// TIA Portal V16 export
// export: Created 2022-11-17T11:55:09.5879993Z, ExportSetting WithDefaults, DisplayName Totally Integrated Automation Portal, DisplayVersion V16 Update 6, DisplayName TIA Portal Version Control Interface, DisplayVersion V16 Update 2, DisplayName TIA Portal Openness, DisplayVersion V16 Update 6, DisplayName SINAMICS Startdrive Advanced, DisplayVersion V16 Update 5, DisplayName SINAMICS Startdrive G130, G150, S120, S150, SINAMICS MV, S210, DisplayVersion V16 Update 5, DisplayName SINAMICS Startdrive G110M, G120, G120C, G120D, G120P, G115D, DisplayVersion V16 Update 5, DisplayName STEP 7 Professional, DisplayVersion V16 Update 6, DisplayName STEP 7 Safety, DisplayVersion V16, DisplayName WinCC Advanced, DisplayVersion V16 Update 6
FUNCTION "FC23_TopTechnoplat" : Void   // FC23, LAD
TITLE = Top Inside
{ S7_Optimized_Access := 'FALSE' }
VERSION : 0.1
// stored: AutoNumber false, IsIECCheckEnabled false, SetENOAutomatically false, UDAEnableTagReadback false
   VAR_TEMP
      LW4 : Word;
   END_VAR
   VAR_TEMP   // added for the SCL form of the ladder/FBD networks
      _w1 : Bool;
      _w2 : Bool;
   END_VAR
BEGIN

REGION Network 1: Top Out Supp. Out - Signal " Top In Position for Pallet Transfe
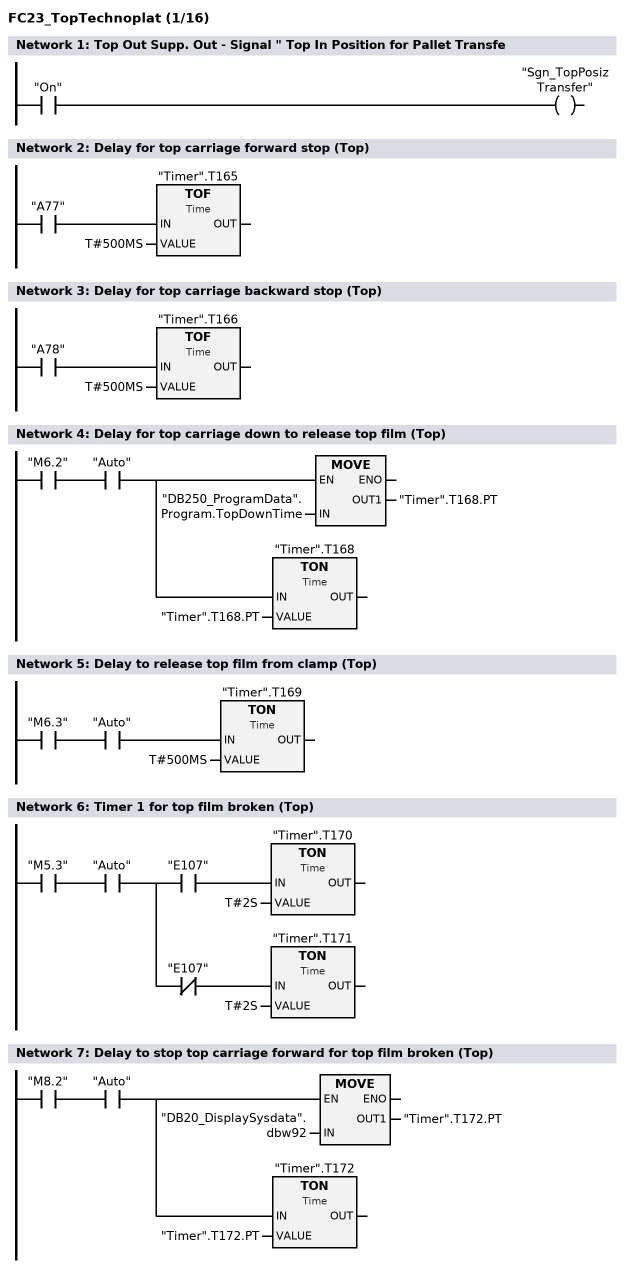
   RUNG wire#powerrail
      Contact( "On" )
      Coil( "Sgn_TopPosizTransfer" )
   END_RUNG
   // the same network as SCL:
   "Sgn_TopPosizTransfer" := "On";
END_REGION

REGION Network 2: Delay for top carriage forward stop (Top)
   "Timer".T165.TOF(IN := "A77", PT := T#500MS);   // TOF coil
END_REGION

REGION Network 3: Delay for top carriage backward stop (Top)
   "Timer".T166.TOF(IN := "A78", PT := T#500MS);   // TOF coil
END_REGION

REGION Network 4: Delay for top carriage down to release top film (Top)
   #_w1 := "M6.2" AND "Auto";
   IF #_w1 THEN "Timer".T168.PT := "DB250_ProgramData".Program.TopDownTime; END_IF;
   "Timer".T168.TON(IN := #_w1, PT := "Timer".T168.PT);   // TON coil
END_REGION

REGION Network 5: Delay to release top film from clamp (Top)
   "Timer".T169.TON(IN := "M6.3" AND "Auto", PT := T#500MS);   // TON coil
END_REGION

REGION Network 6: Timer 1 for top film broken (Top)
   #_w1 := "M5.3" AND "Auto";
   "Timer".T170.TON(IN := #_w1 AND "E107", PT := T#2S);   // TON coil
   "Timer".T171.TON(IN := #_w1 AND NOT "E107", PT := T#2S);   // TON coil
END_REGION

REGION Network 7: Delay to stop top carriage forward for top film broken (Top)
   #_w1 := "M8.2" AND "Auto";
   IF #_w1 THEN "Timer".T172.PT := "DB20_DisplaySysdata".dbw92; END_IF;
   "Timer".T172.TON(IN := #_w1, PT := "Timer".T172.PT);   // TON coil
END_REGION

REGION Network 8: Delay to stop top carriage against vibration (Top)
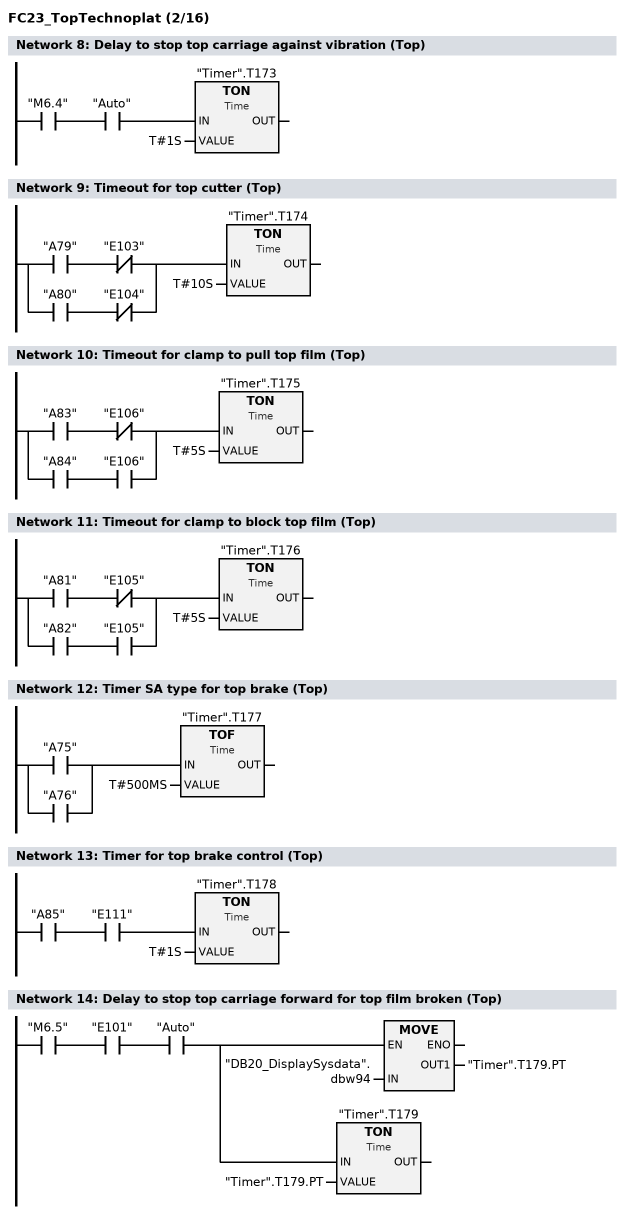
   "Timer".T173.TON(IN := "M6.4" AND "Auto", PT := T#1S);   // TON coil
END_REGION

REGION Network 9: Timeout for top cutter (Top)
   "Timer".T174.TON(IN := ("A79" AND NOT "E103") OR ("A80" AND NOT "E104"), PT := T#10S);   // TON coil
END_REGION

REGION Network 10: Timeout for clamp to pull top film (Top)
   "Timer".T175.TON(IN := ("A83" AND NOT "E106") OR ("A84" AND "E106"), PT := T#5S);   // TON coil
END_REGION

REGION Network 11: Timeout for clamp to block top film (Top)
   "Timer".T176.TON(IN := ("A81" AND NOT "E105") OR ("A82" AND "E105"), PT := T#5S);   // TON coil
END_REGION

REGION Network 12: Timer SA type for top brake (Top)
   "Timer".T177.TOF(IN := "A75" OR "A76", PT := T#500MS);   // TOF coil
END_REGION

REGION Network 13: Timer for top brake control (Top)
   "Timer".T178.TON(IN := "A85" AND "E111", PT := T#1S);   // TON coil
END_REGION

REGION Network 14: Delay to stop top carriage forward for top film broken (Top)
   #_w1 := "M6.5" AND "E101" AND "Auto";
   IF #_w1 THEN "Timer".T179.PT := "DB20_DisplaySysdata".dbw94; END_IF;
   "Timer".T179.TON(IN := #_w1, PT := "Timer".T179.PT);   // TON coil
END_REGION

REGION Network 15: Carriage in position to rotate in medium to wrap top
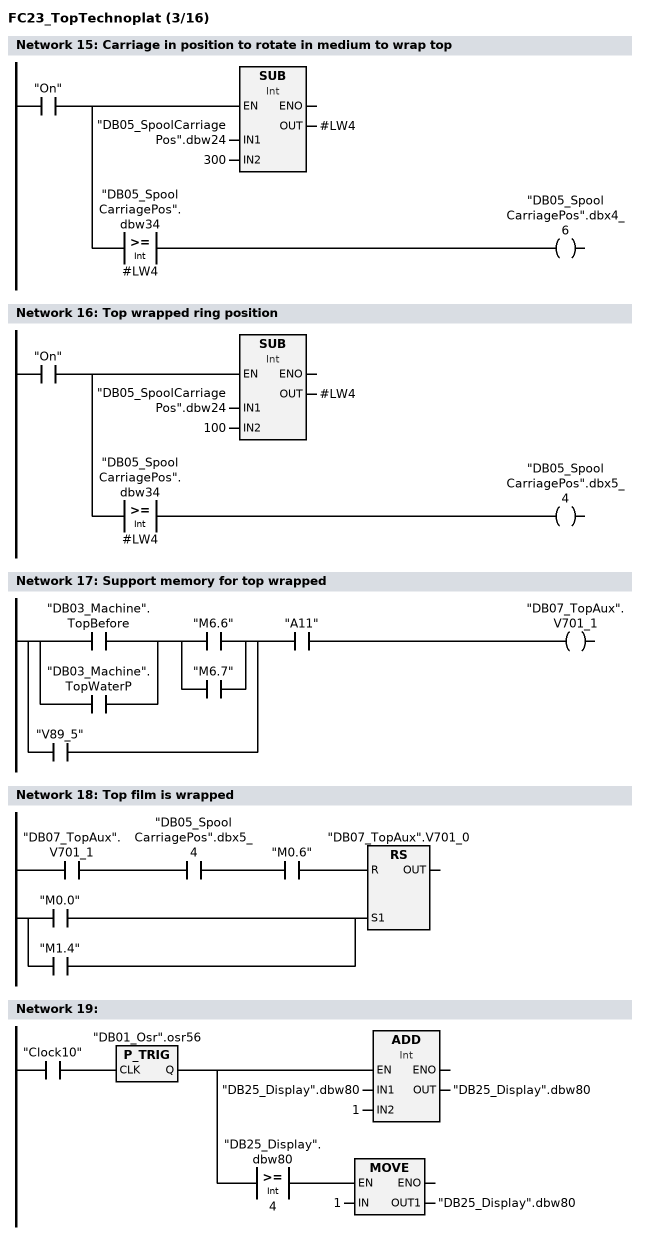
   RUNG wire#powerrail
      Contact( "On" )
      wire#w1
      { S7_Templates := "SrcType := Int"; S7_GenerateENO := "TRUE" } Sub(in1 := "DB05_SpoolCarriagePos".dbw24, in2 := 300, out => #LW4)
   END_RUNG
   RUNG wire#w1
      { S7_Templates := "SrcType := Int" } GE_Contact(in1 := "DB05_SpoolCarriagePos".dbw34, in2 := #LW4)
      Coil( "DB05_SpoolCarriagePos".dbx4_6 )
   END_RUNG
   // the same network as SCL:
   IF "On" THEN #LW4 := "DB05_SpoolCarriagePos".dbw24 - 300; END_IF;
   "DB05_SpoolCarriagePos".dbx4_6 := "On" AND ("DB05_SpoolCarriagePos".dbw34 >= #LW4);
END_REGION

REGION Network 16: Top wrapped ring position
   RUNG wire#powerrail
      Contact( "On" )
      wire#w1
      { S7_Templates := "SrcType := Int"; S7_GenerateENO := "TRUE" } Sub(in1 := "DB05_SpoolCarriagePos".dbw24, in2 := 100, out => #LW4)
   END_RUNG
   RUNG wire#w1
      { S7_Templates := "SrcType := Int" } GE_Contact(in1 := "DB05_SpoolCarriagePos".dbw34, in2 := #LW4)
      Coil( "DB05_SpoolCarriagePos".dbx5_4 )
   END_RUNG
   // the same network as SCL:
   IF "On" THEN #LW4 := "DB05_SpoolCarriagePos".dbw24 - 100; END_IF;
   "DB05_SpoolCarriagePos".dbx5_4 := "On" AND ("DB05_SpoolCarriagePos".dbw34 >= #LW4);
END_REGION

REGION Network 17: Support memory for top wrapped
   RUNG wire#powerrail
      Contact( "DB03_Machine".TopBefore )
      wire#w1
      Contact( "M6.6" )
      wire#w2
      Contact( "A11" )
      Coil( "DB07_TopAux".V701_1 )
   END_RUNG
   RUNG wire#powerrail
      Contact( "DB03_Machine".TopWaterP )
   END_RUNG wire#w1
   RUNG wire#w1
      Contact( "M6.7" )
   END_RUNG wire#w2
   RUNG wire#powerrail
      Contact( "V89_5" )
   END_RUNG wire#w2
   // the same network as SCL:
   "DB07_TopAux".V701_1 := ((("DB03_Machine".TopBefore OR "DB03_Machine".TopWaterP) AND ("M6.6" OR "M6.7")) OR "V89_5") AND "A11";
END_REGION

REGION Network 18: Top film is wrapped
   RUNG wire#powerrail
      Contact( "DB07_TopAux".V701_1 )
      Contact( "DB05_SpoolCarriagePos".dbx5_4 )
      Contact( "M0.6" )
      S_RS(operand := "DB07_TopAux".V701_0, s1 := wire#w1)
   END_RUNG
   RUNG wire#powerrail
      Contact( "M0.0" )
   END_RUNG wire#w1
   RUNG wire#powerrail
      Contact( "M1.4" )
   END_RUNG wire#w1
   // the same network as SCL:
   IF "DB07_TopAux".V701_1 AND "DB05_SpoolCarriagePos".dbx5_4 AND "M0.6" THEN
       "DB07_TopAux".V701_0 := FALSE;   // RS flip-flop
   END_IF;
   IF "M0.0" OR "M1.4" THEN "DB07_TopAux".V701_0 := TRUE; END_IF;
END_REGION

REGION Network 19
   RUNG wire#powerrail
      Contact( "Clock10" )
      P_Trig( "DB01_Osr".osr56 )
      wire#w1
      { S7_Templates := "SrcType := Int"; S7_GenerateENO := "TRUE" } Add(in1 := "DB25_Display".dbw80, in2 := 1, out => "DB25_Display".dbw80)
   END_RUNG
   RUNG wire#w1
      { S7_Templates := "SrcType := Int" } GE_Contact(in1 := "DB25_Display".dbw80, in2 := 4)
      { S7_GenerateENO := "TRUE" } Move(in := 1, out1 => "DB25_Display".dbw80)
   END_RUNG
   // the same network as SCL:
   #_w1 := "Clock10" AND NOT "DB01_Osr".osr56;   // rising edge
   "DB01_Osr".osr56 := "Clock10";
   IF #_w1 THEN "DB25_Display".dbw80 := "DB25_Display".dbw80 + 1; END_IF;
   IF #_w1 AND ("DB25_Display".dbw80 >= 4) THEN "DB25_Display".dbw80 := 1; END_IF;
END_REGION

REGION Network 20: Arm rotation speed: Middle 1 for top
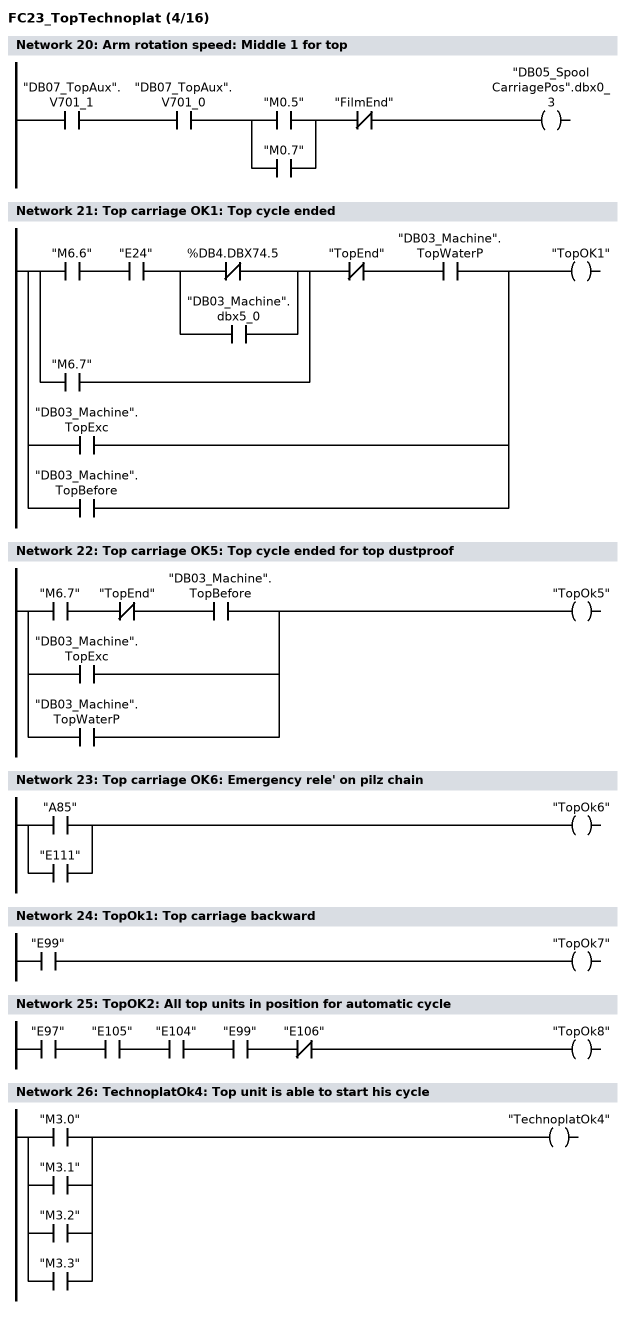
   RUNG wire#powerrail
      Contact( "DB07_TopAux".V701_1 )
      Contact( "DB07_TopAux".V701_0 )
      wire#w1
      Contact( "M0.5" )
      wire#w2
      I_Contact( "FilmEnd" )
      Coil( "DB05_SpoolCarriagePos".dbx0_3 )
   END_RUNG
   RUNG wire#w1
      Contact( "M0.7" )
   END_RUNG wire#w2
   // the same network as SCL:
   "DB05_SpoolCarriagePos".dbx0_3 := "DB07_TopAux".V701_1 AND "DB07_TopAux".V701_0 AND ("M0.5" OR "M0.7") AND NOT "FilmEnd";
END_REGION

REGION Network 21: Top carriage OK1: Top cycle ended
   RUNG wire#powerrail
      Contact( "M6.6" )
      Contact( "E24" )
      wire#w1
      I_Contact( %DB4.DBX74.5 )
      wire#w2
      I_Contact( "TopEnd" )
      Contact( "DB03_Machine".TopWaterP )
      wire#w3
      Coil( "TopOK1" )
   END_RUNG
   RUNG wire#w1
      Contact( "DB03_Machine".dbx5_0 )
   END_RUNG wire#w2
   RUNG wire#powerrail
      Contact( "M6.7" )
   END_RUNG wire#w2
   RUNG wire#powerrail
      Contact( "DB03_Machine".TopExc )
   END_RUNG wire#w3
   RUNG wire#powerrail
      Contact( "DB03_Machine".TopBefore )
   END_RUNG wire#w3
   // the same network as SCL:
   "TopOK1" := ((("M6.6" AND "E24" AND (NOT %DB4.DBX74.5 OR "DB03_Machine".dbx5_0)) OR "M6.7") AND NOT "TopEnd" AND "DB03_Machine".TopWaterP) OR "DB03_Machine".TopExc OR "DB03_Machine".TopBefore;
END_REGION

REGION Network 22: Top carriage OK5: Top cycle ended for top dustproof
   RUNG wire#powerrail
      Contact( "M6.7" )
      I_Contact( "TopEnd" )
      Contact( "DB03_Machine".TopBefore )
      wire#w1
      Coil( "TopOk5" )
   END_RUNG
   RUNG wire#powerrail
      Contact( "DB03_Machine".TopExc )
   END_RUNG wire#w1
   RUNG wire#powerrail
      Contact( "DB03_Machine".TopWaterP )
   END_RUNG wire#w1
   // the same network as SCL:
   "TopOk5" := ("M6.7" AND NOT "TopEnd" AND "DB03_Machine".TopBefore) OR "DB03_Machine".TopExc OR "DB03_Machine".TopWaterP;
END_REGION

REGION Network 23: Top carriage OK6: Emergency rele' on pilz chain
   RUNG wire#powerrail
      Contact( "A85" )
      wire#w1
      Coil( "TopOk6" )
   END_RUNG
   RUNG wire#powerrail
      Contact( "E111" )
   END_RUNG wire#w1
   // the same network as SCL:
   "TopOk6" := "A85" OR "E111";
END_REGION

REGION Network 24: TopOk1: Top carriage backward
   RUNG wire#powerrail
      Contact( "E99" )
      Coil( "TopOk7" )
   END_RUNG
   // the same network as SCL:
   "TopOk7" := "E99";
END_REGION

REGION Network 25: TopOK2: All top units in position for automatic cycle
   RUNG wire#powerrail
      Contact( "E97" )
      Contact( "E105" )
      Contact( "E104" )
      Contact( "E99" )
      I_Contact( "E106" )
      Coil( "TopOk8" )
   END_RUNG
   // the same network as SCL:
   "TopOk8" := "E97" AND "E105" AND "E104" AND "E99" AND NOT "E106";
END_REGION

REGION Network 26: TechnoplatOk4: Top unit is able to start his cycle
   RUNG wire#powerrail
      Contact( "M3.0" )
      wire#w1
      Coil( "TechnoplatOk4" )
   END_RUNG
   RUNG wire#powerrail
      Contact( "M3.1" )
   END_RUNG wire#w1
   RUNG wire#powerrail
      Contact( "M3.2" )
   END_RUNG wire#w1
   RUNG wire#powerrail
      Contact( "M3.3" )
   END_RUNG wire#w1
   // the same network as SCL:
   "TechnoplatOk4" := "M3.0" OR "M3.1" OR "M3.2" OR "M3.3";
END_REGION

REGION Network 27: Top film ended or broken
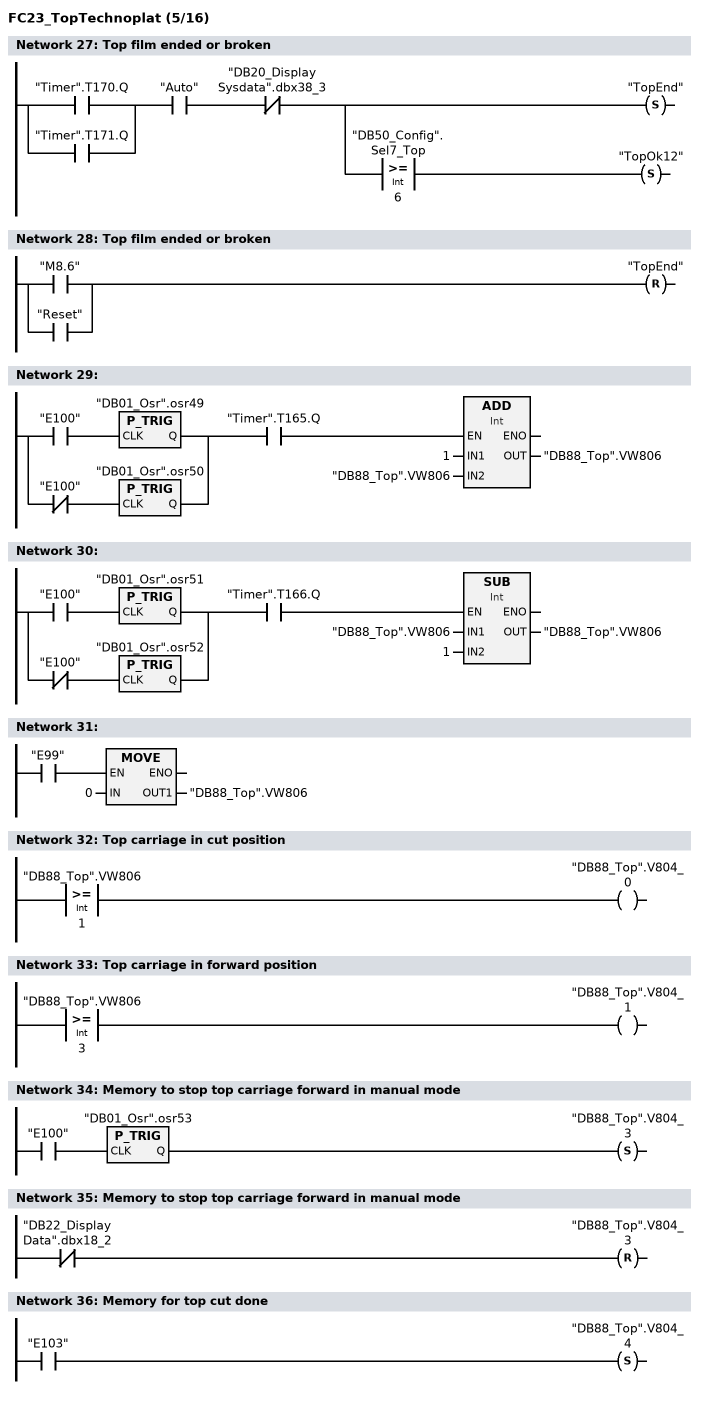
   RUNG wire#powerrail
      Contact( "Timer".T170.Q )
      wire#w1
      Contact( "Auto" )
      I_Contact( "DB20_DisplaySysdata".dbx38_3 )
      wire#w2
      S_Coil( "TopEnd" )
   END_RUNG
   RUNG wire#powerrail
      Contact( "Timer".T171.Q )
   END_RUNG wire#w1
   RUNG wire#w2
      { S7_Templates := "SrcType := Int" } GE_Contact(in1 := "DB50_Config".Sel7_Top, in2 := 6)
      S_Coil( "TopOk12" )
   END_RUNG
   // the same network as SCL:
   #_w1 := ("Timer".T170.Q OR "Timer".T171.Q) AND "Auto" AND NOT "DB20_DisplaySysdata".dbx38_3;
   IF #_w1 THEN "TopEnd" := TRUE; END_IF;
   IF #_w1 AND ("DB50_Config".Sel7_Top >= 6) THEN "TopOk12" := TRUE; END_IF;
END_REGION

REGION Network 28: Top film ended or broken
   RUNG wire#powerrail
      Contact( "M8.6" )
      wire#w1
      R_Coil( "TopEnd" )
   END_RUNG
   RUNG wire#powerrail
      Contact( "Reset" )
   END_RUNG wire#w1
   // the same network as SCL:
   IF "M8.6" OR "Reset" THEN "TopEnd" := FALSE; END_IF;
END_REGION

REGION Network 29
   RUNG wire#powerrail
      Contact( "E100" )
      P_Trig( "DB01_Osr".osr49 )
      wire#w1
      Contact( "Timer".T165.Q )
      { S7_Templates := "SrcType := Int"; S7_GenerateENO := "TRUE" } Add(in1 := 1, in2 := "DB88_Top".VW806, out => "DB88_Top".VW806)
   END_RUNG
   RUNG wire#powerrail
      I_Contact( "E100" )
      P_Trig( "DB01_Osr".osr50 )
   END_RUNG wire#w1
   // the same network as SCL:
   #_w1 := "E100" AND NOT "DB01_Osr".osr49;   // rising edge
   "DB01_Osr".osr49 := "E100";
   #_w2 := NOT "E100" AND NOT "DB01_Osr".osr50;   // rising edge
   "DB01_Osr".osr50 := NOT "E100";
   IF (#_w1 OR #_w2) AND "Timer".T165.Q THEN "DB88_Top".VW806 := 1 + "DB88_Top".VW806; END_IF;
END_REGION

REGION Network 30
   RUNG wire#powerrail
      Contact( "E100" )
      P_Trig( "DB01_Osr".osr51 )
      wire#w1
      Contact( "Timer".T166.Q )
      { S7_Templates := "SrcType := Int"; S7_GenerateENO := "TRUE" } Sub(in1 := "DB88_Top".VW806, in2 := 1, out => "DB88_Top".VW806)
   END_RUNG
   RUNG wire#powerrail
      I_Contact( "E100" )
      P_Trig( "DB01_Osr".osr52 )
   END_RUNG wire#w1
   // the same network as SCL:
   #_w1 := "E100" AND NOT "DB01_Osr".osr51;   // rising edge
   "DB01_Osr".osr51 := "E100";
   #_w2 := NOT "E100" AND NOT "DB01_Osr".osr52;   // rising edge
   "DB01_Osr".osr52 := NOT "E100";
   IF (#_w1 OR #_w2) AND "Timer".T166.Q THEN "DB88_Top".VW806 := "DB88_Top".VW806 - 1; END_IF;
END_REGION

REGION Network 31
   RUNG wire#powerrail
      Contact( "E99" )
      { S7_GenerateENO := "TRUE" } Move(in := 0, out1 => "DB88_Top".VW806)
   END_RUNG
   // the same network as SCL:
   IF "E99" THEN "DB88_Top".VW806 := 0; END_IF;
END_REGION

REGION Network 32: Top carriage in cut position
   RUNG wire#powerrail
      { S7_Templates := "SrcType := Int" } GE_Contact(in1 := "DB88_Top".VW806, in2 := 1)
      Coil( "DB88_Top".V804_0 )
   END_RUNG
   // the same network as SCL:
   "DB88_Top".V804_0 := "DB88_Top".VW806 >= 1;
END_REGION

REGION Network 33: Top carriage in forward position
   RUNG wire#powerrail
      { S7_Templates := "SrcType := Int" } GE_Contact(in1 := "DB88_Top".VW806, in2 := 3)
      Coil( "DB88_Top".V804_1 )
   END_RUNG
   // the same network as SCL:
   "DB88_Top".V804_1 := "DB88_Top".VW806 >= 3;
END_REGION

REGION Network 34: Memory to stop top carriage forward in manual mode
   RUNG wire#powerrail
      Contact( "E100" )
      P_Trig( "DB01_Osr".osr53 )
      S_Coil( "DB88_Top".V804_3 )
   END_RUNG
   // the same network as SCL:
   #_w1 := "E100" AND NOT "DB01_Osr".osr53;   // rising edge
   "DB01_Osr".osr53 := "E100";
   IF #_w1 THEN "DB88_Top".V804_3 := TRUE; END_IF;
END_REGION

REGION Network 35: Memory to stop top carriage forward in manual mode
   RUNG wire#powerrail
      I_Contact( "DB22_DisplayData".dbx18_2 )
      R_Coil( "DB88_Top".V804_3 )
   END_RUNG
   // the same network as SCL:
   IF NOT "DB22_DisplayData".dbx18_2 THEN "DB88_Top".V804_3 := FALSE; END_IF;
END_REGION

REGION Network 36: Memory for top cut done
   RUNG wire#powerrail
      Contact( "E103" )
      S_Coil( "DB88_Top".V804_4 )
   END_RUNG
   // the same network as SCL:
   IF "E103" THEN "DB88_Top".V804_4 := TRUE; END_IF;
END_REGION

REGION Network 37: Memory for top cut done
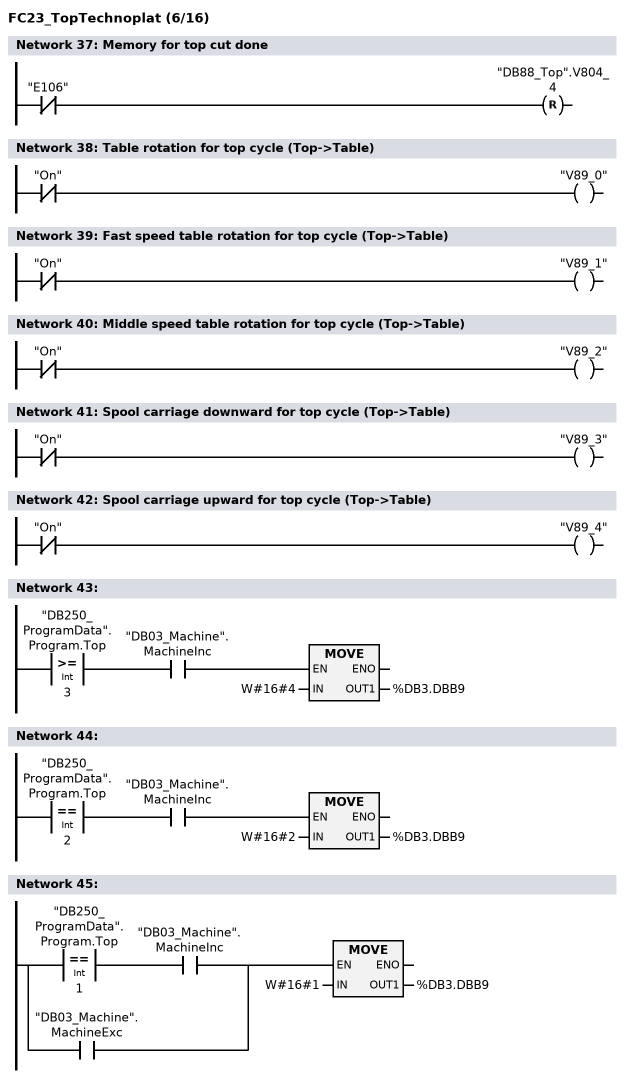
   RUNG wire#powerrail
      I_Contact( "E106" )
      R_Coil( "DB88_Top".V804_4 )
   END_RUNG
   // the same network as SCL:
   IF NOT "E106" THEN "DB88_Top".V804_4 := FALSE; END_IF;
END_REGION

REGION Network 38: Table rotation for top cycle (Top->Table)
   RUNG wire#powerrail
      I_Contact( "On" )
      Coil( "V89_0" )
   END_RUNG
   // the same network as SCL:
   "V89_0" := NOT "On";
END_REGION

REGION Network 39: Fast speed table rotation for top cycle (Top->Table)
   RUNG wire#powerrail
      I_Contact( "On" )
      Coil( "V89_1" )
   END_RUNG
   // the same network as SCL:
   "V89_1" := NOT "On";
END_REGION

REGION Network 40: Middle speed table rotation for top cycle (Top->Table)
   RUNG wire#powerrail
      I_Contact( "On" )
      Coil( "V89_2" )
   END_RUNG
   // the same network as SCL:
   "V89_2" := NOT "On";
END_REGION

REGION Network 41: Spool carriage downward for top cycle (Top->Table)
   RUNG wire#powerrail
      I_Contact( "On" )
      Coil( "V89_3" )
   END_RUNG
   // the same network as SCL:
   "V89_3" := NOT "On";
END_REGION

REGION Network 42: Spool carriage upward for top cycle (Top->Table)
   RUNG wire#powerrail
      I_Contact( "On" )
      Coil( "V89_4" )
   END_RUNG
   // the same network as SCL:
   "V89_4" := NOT "On";
END_REGION

REGION Network 43
   RUNG wire#powerrail
      { S7_Templates := "SrcType := Int" } GE_Contact(in1 := "DB250_ProgramData".Program.Top, in2 := 3)
      Contact( "DB03_Machine".MachineInc )
      { S7_GenerateENO := "TRUE" } Move(in := W#16#4, out1 => %DB3.DBB9)
   END_RUNG
   // the same network as SCL:
   IF ("DB250_ProgramData".Program.Top >= 3) AND "DB03_Machine".MachineInc THEN %DB3.DBB9 := W#16#4; END_IF;
END_REGION

REGION Network 44
   RUNG wire#powerrail
      { S7_Templates := "SrcType := Int" } EQ_Contact(in1 := "DB250_ProgramData".Program.Top, in2 := 2)
      Contact( "DB03_Machine".MachineInc )
      { S7_GenerateENO := "TRUE" } Move(in := W#16#2, out1 => %DB3.DBB9)
   END_RUNG
   // the same network as SCL:
   IF ("DB250_ProgramData".Program.Top = 2) AND "DB03_Machine".MachineInc THEN %DB3.DBB9 := W#16#2; END_IF;
END_REGION

REGION Network 45
   RUNG wire#powerrail
      { S7_Templates := "SrcType := Int" } EQ_Contact(in1 := "DB250_ProgramData".Program.Top, in2 := 1)
      Contact( "DB03_Machine".MachineInc )
      wire#w1
      { S7_GenerateENO := "TRUE" } Move(in := W#16#1, out1 => %DB3.DBB9)
   END_RUNG
   RUNG wire#powerrail
      Contact( "DB03_Machine".MachineExc )
   END_RUNG wire#w1
   // the same network as SCL:
   IF (("DB250_ProgramData".Program.Top = 1) AND "DB03_Machine".MachineInc) OR "DB03_Machine".MachineExc THEN
       %DB3.DBB9 := W#16#1;
   END_IF;
END_REGION

REGION Network 46: Wrapping cycle: After this step top waterproof
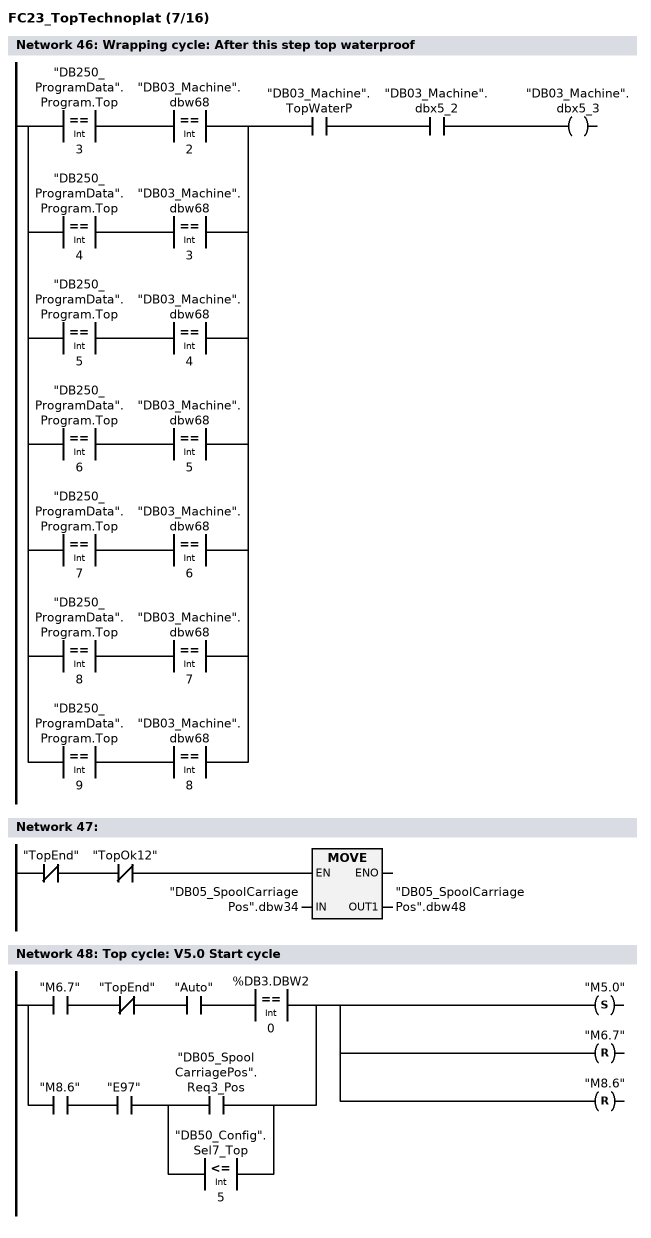
   RUNG wire#powerrail
      { S7_Templates := "SrcType := Int" } EQ_Contact(in1 := "DB250_ProgramData".Program.Top, in2 := 3)
      { S7_Templates := "SrcType := Int" } EQ_Contact(in1 := "DB03_Machine".dbw68, in2 := 2)
      wire#w1
      Contact( "DB03_Machine".TopWaterP )
      Contact( "DB03_Machine".dbx5_2 )
      Coil( "DB03_Machine".dbx5_3 )
   END_RUNG
   RUNG wire#powerrail
      { S7_Templates := "SrcType := Int" } EQ_Contact(in1 := "DB250_ProgramData".Program.Top, in2 := 4)
      { S7_Templates := "SrcType := Int" } EQ_Contact(in1 := "DB03_Machine".dbw68, in2 := 3)
   END_RUNG wire#w1
   RUNG wire#powerrail
      { S7_Templates := "SrcType := Int" } EQ_Contact(in1 := "DB250_ProgramData".Program.Top, in2 := 5)
      { S7_Templates := "SrcType := Int" } EQ_Contact(in1 := "DB03_Machine".dbw68, in2 := 4)
   END_RUNG wire#w1
   RUNG wire#powerrail
      { S7_Templates := "SrcType := Int" } EQ_Contact(in1 := "DB250_ProgramData".Program.Top, in2 := 6)
      { S7_Templates := "SrcType := Int" } EQ_Contact(in1 := "DB03_Machine".dbw68, in2 := 5)
   END_RUNG wire#w1
   RUNG wire#powerrail
      { S7_Templates := "SrcType := Int" } EQ_Contact(in1 := "DB250_ProgramData".Program.Top, in2 := 7)
      { S7_Templates := "SrcType := Int" } EQ_Contact(in1 := "DB03_Machine".dbw68, in2 := 6)
   END_RUNG wire#w1
   RUNG wire#powerrail
      { S7_Templates := "SrcType := Int" } EQ_Contact(in1 := "DB250_ProgramData".Program.Top, in2 := 8)
      { S7_Templates := "SrcType := Int" } EQ_Contact(in1 := "DB03_Machine".dbw68, in2 := 7)
   END_RUNG wire#w1
   RUNG wire#powerrail
      { S7_Templates := "SrcType := Int" } EQ_Contact(in1 := "DB250_ProgramData".Program.Top, in2 := 9)
      { S7_Templates := "SrcType := Int" } EQ_Contact(in1 := "DB03_Machine".dbw68, in2 := 8)
   END_RUNG wire#w1
   // the same network as SCL:
   "DB03_Machine".dbx5_3 := ((("DB250_ProgramData".Program.Top = 3) AND ("DB03_Machine".dbw68 = 2)) OR (("DB250_ProgramData".Program.Top = 4) AND ("DB03_Machine".dbw68 = 3)) OR (("DB250_ProgramData".Program.Top = 5) AND ("DB03_Machine".dbw68 = 4)) OR (("DB250_ProgramData".Program.Top = 6) AND ("DB03_Machine".dbw68 = 5)) OR (("DB250_ProgramData".Program.Top = 7) AND ("DB03_Machine".dbw68 = 6)) OR (("DB250_ProgramData".Program.Top = 8) AND ("DB03_Machine".dbw68 = 7)) OR (("DB250_ProgramData".Program.Top = 9) AND ("DB03_Machine".dbw68 = 8))) AND "DB03_Machine".TopWaterP AND "DB03_Machine".dbx5_2;
END_REGION

REGION Network 47
   RUNG wire#powerrail
      I_Contact( "TopEnd" )
      I_Contact( "TopOk12" )
      { S7_GenerateENO := "TRUE" } Move(in := "DB05_SpoolCarriagePos".dbw34, out1 => "DB05_SpoolCarriagePos".dbw48)
   END_RUNG
   // the same network as SCL:
   IF NOT "TopEnd" AND NOT "TopOk12" THEN
       "DB05_SpoolCarriagePos".dbw48 := "DB05_SpoolCarriagePos".dbw34;
   END_IF;
END_REGION

REGION Network 48: Top cycle: V5.0 Start cycle
   RUNG wire#powerrail
      Contact( "M6.7" )
      I_Contact( "TopEnd" )
      Contact( "Auto" )
      { S7_Templates := "SrcType := Int" } EQ_Contact(in1 := %DB3.DBW2, in2 := 0)
      wire#w1
      S_Coil( "M5.0" )
   END_RUNG
   RUNG wire#powerrail
      Contact( "M8.6" )
      Contact( "E97" )
      wire#w2
      Contact( "DB05_SpoolCarriagePos".Req3_Pos )
   END_RUNG wire#w1
   RUNG wire#w2
      { S7_Templates := "SrcType := Int" } LE_Contact(in1 := "DB50_Config".Sel7_Top, in2 := 5)
   END_RUNG wire#w1
   RUNG wire#w1
      R_Coil( "M6.7" )
   END_RUNG
   RUNG wire#w1
      R_Coil( "M8.6" )
   END_RUNG
   // the same network as SCL:
   IF ("M6.7" AND NOT "TopEnd" AND "Auto" AND (%DB3.DBW2 = 0)) OR ("M8.6" AND "E97" AND ("DB05_SpoolCarriagePos".Req3_Pos OR ("DB50_Config".Sel7_Top <= 5))) THEN
       "M5.0" := TRUE;
   END_IF;
   #_w1 := ("M6.7" AND NOT "TopEnd" AND "Auto" AND (%DB3.DBW2 = 0)) OR ("M8.6" AND "E97" AND ("DB05_SpoolCarriagePos".Req3_Pos OR ("DB50_Config".Sel7_Top <= 5)));
   IF #_w1 THEN
       "M6.7" := FALSE;
       "M8.6" := FALSE;
   END_IF;
END_REGION

REGION Network 49: Top cycle: V5.1 Closing clamp to pull top film
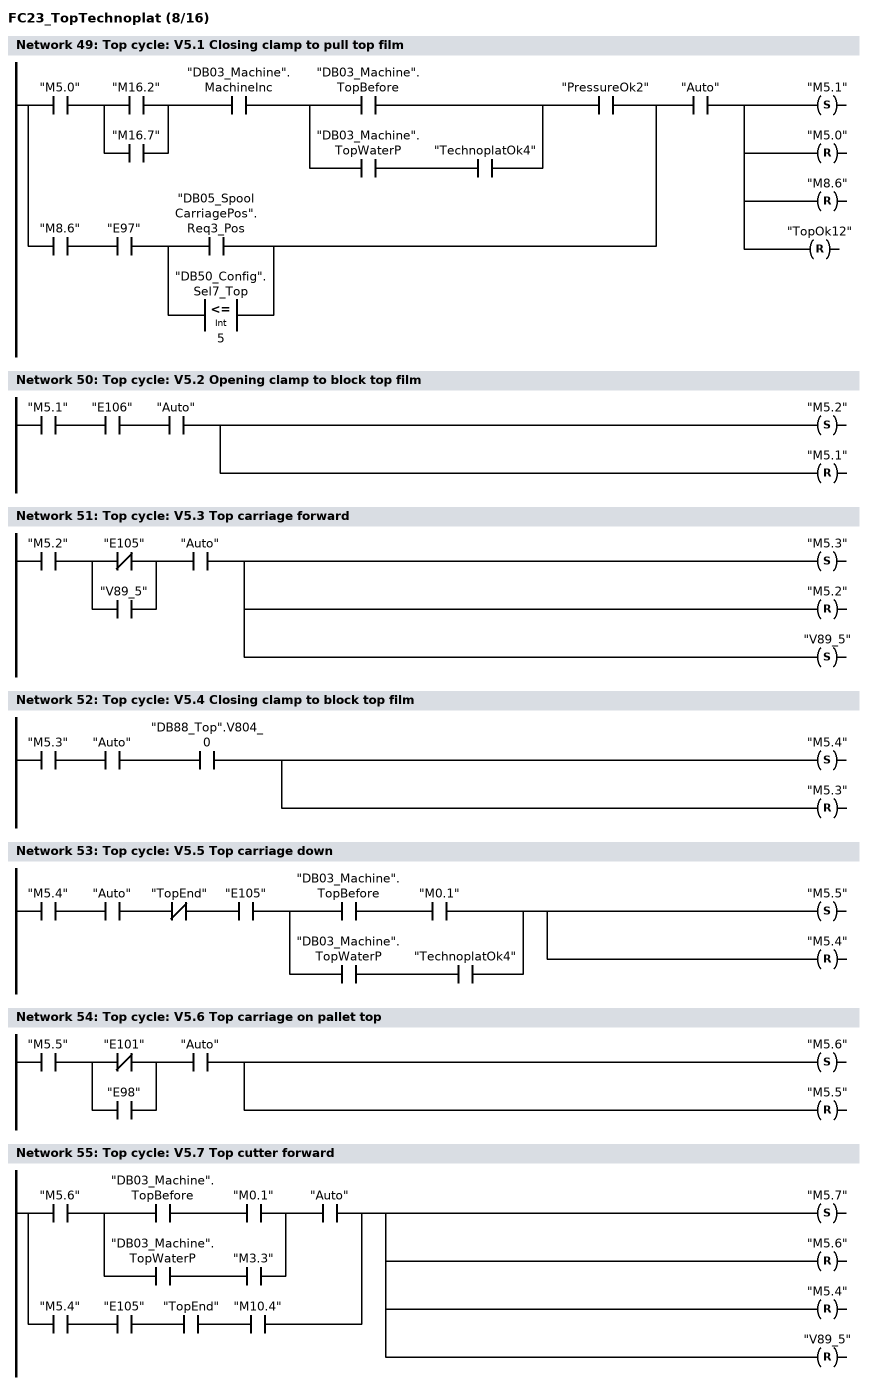
   RUNG wire#powerrail
      Contact( "M5.0" )
      wire#w1
      Contact( "M16.2" )
      wire#w2
      Contact( "DB03_Machine".MachineInc )
      wire#w3
      Contact( "DB03_Machine".TopBefore )
      wire#w4
      Contact( "PressureOk2" )
      wire#w5
      Contact( "Auto" )
      wire#w7
      S_Coil( "M5.1" )
   END_RUNG
   RUNG wire#w1
      Contact( "M16.7" )
   END_RUNG wire#w2
   RUNG wire#w3
      Contact( "DB03_Machine".TopWaterP )
      Contact( "TechnoplatOk4" )
   END_RUNG wire#w4
   RUNG wire#powerrail
      Contact( "M8.6" )
      Contact( "E97" )
      wire#w6
      Contact( "DB05_SpoolCarriagePos".Req3_Pos )
   END_RUNG wire#w5
   RUNG wire#w6
      { S7_Templates := "SrcType := Int" } LE_Contact(in1 := "DB50_Config".Sel7_Top, in2 := 5)
   END_RUNG wire#w5
   RUNG wire#w7
      R_Coil( "M5.0" )
   END_RUNG
   RUNG wire#w7
      R_Coil( "M8.6" )
   END_RUNG
   RUNG wire#w7
      R_Coil( "TopOk12" )
   END_RUNG
   // the same network as SCL:
   IF (("M5.0" AND ("M16.2" OR "M16.7") AND "DB03_Machine".MachineInc AND ("DB03_Machine".TopBefore OR ("DB03_Machine".TopWaterP AND "TechnoplatOk4")) AND "PressureOk2") OR ("M8.6" AND "E97" AND ("DB05_SpoolCarriagePos".Req3_Pos OR ("DB50_Config".Sel7_Top <= 5)))) AND "Auto" THEN
       "M5.1" := TRUE;
   END_IF;
   #_w1 := (("M5.0" AND ("M16.2" OR "M16.7") AND "DB03_Machine".MachineInc AND ("DB03_Machine".TopBefore OR ("DB03_Machine".TopWaterP AND "TechnoplatOk4")) AND "PressureOk2") OR ("M8.6" AND "E97" AND ("DB05_SpoolCarriagePos".Req3_Pos OR ("DB50_Config".Sel7_Top <= 5)))) AND "Auto";
   IF #_w1 THEN
       "M5.0" := FALSE;
       "M8.6" := FALSE;
       "TopOk12" := FALSE;
   END_IF;
END_REGION

REGION Network 50: Top cycle: V5.2 Opening clamp to block top film
   RUNG wire#powerrail
      Contact( "M5.1" )
      Contact( "E106" )
      Contact( "Auto" )
      wire#w1
      S_Coil( "M5.2" )
   END_RUNG
   RUNG wire#w1
      R_Coil( "M5.1" )
   END_RUNG
   // the same network as SCL:
   IF "M5.1" AND "E106" AND "Auto" THEN
       "M5.2" := TRUE;
       "M5.1" := FALSE;
   END_IF;
END_REGION

REGION Network 51: Top cycle: V5.3 Top carriage forward
   RUNG wire#powerrail
      Contact( "M5.2" )
      wire#w1
      I_Contact( "E105" )
      wire#w2
      Contact( "Auto" )
      wire#w3
      S_Coil( "M5.3" )
   END_RUNG
   RUNG wire#w1
      Contact( "V89_5" )
   END_RUNG wire#w2
   RUNG wire#w3
      R_Coil( "M5.2" )
   END_RUNG
   RUNG wire#w3
      S_Coil( "V89_5" )
   END_RUNG
   // the same network as SCL:
   IF "M5.2" AND (NOT "E105" OR "V89_5") AND "Auto" THEN "M5.3" := TRUE; END_IF;
   #_w1 := "M5.2" AND (NOT "E105" OR "V89_5") AND "Auto";
   IF #_w1 THEN
       "M5.2" := FALSE;
       "V89_5" := TRUE;
   END_IF;
END_REGION

REGION Network 52: Top cycle: V5.4 Closing clamp to block top film
   RUNG wire#powerrail
      Contact( "M5.3" )
      Contact( "Auto" )
      Contact( "DB88_Top".V804_0 )
      wire#w1
      S_Coil( "M5.4" )
   END_RUNG
   RUNG wire#w1
      R_Coil( "M5.3" )
   END_RUNG
   // the same network as SCL:
   IF "M5.3" AND "Auto" AND "DB88_Top".V804_0 THEN
       "M5.4" := TRUE;
       "M5.3" := FALSE;
   END_IF;
END_REGION

REGION Network 53: Top cycle: V5.5 Top carriage down
   RUNG wire#powerrail
      Contact( "M5.4" )
      Contact( "Auto" )
      I_Contact( "TopEnd" )
      Contact( "E105" )
      wire#w1
      Contact( "DB03_Machine".TopBefore )
      Contact( "M0.1" )
      wire#w2
      S_Coil( "M5.5" )
   END_RUNG
   RUNG wire#w1
      Contact( "DB03_Machine".TopWaterP )
      Contact( "TechnoplatOk4" )
   END_RUNG wire#w2
   RUNG wire#w2
      R_Coil( "M5.4" )
   END_RUNG
   // the same network as SCL:
   IF "M5.4" AND "Auto" AND NOT "TopEnd" AND "E105" AND (("DB03_Machine".TopBefore AND "M0.1") OR ("DB03_Machine".TopWaterP AND "TechnoplatOk4")) THEN
       "M5.5" := TRUE;
       "M5.4" := FALSE;
   END_IF;
END_REGION

REGION Network 54: Top cycle: V5.6 Top carriage on pallet top
   RUNG wire#powerrail
      Contact( "M5.5" )
      wire#w1
      I_Contact( "E101" )
      wire#w2
      Contact( "Auto" )
      wire#w3
      S_Coil( "M5.6" )
   END_RUNG
   RUNG wire#w1
      Contact( "E98" )
   END_RUNG wire#w2
   RUNG wire#w3
      R_Coil( "M5.5" )
   END_RUNG
   // the same network as SCL:
   IF "M5.5" AND (NOT "E101" OR "E98") AND "Auto" THEN
       "M5.6" := TRUE;
       "M5.5" := FALSE;
   END_IF;
END_REGION

REGION Network 55: Top cycle: V5.7 Top cutter forward
   RUNG wire#powerrail
      Contact( "M5.6" )
      wire#w1
      Contact( "DB03_Machine".TopBefore )
      Contact( "M0.1" )
      wire#w2
      Contact( "Auto" )
      wire#w3
      S_Coil( "M5.7" )
   END_RUNG
   RUNG wire#w1
      Contact( "DB03_Machine".TopWaterP )
      Contact( "M3.3" )
   END_RUNG wire#w2
   RUNG wire#powerrail
      Contact( "M5.4" )
      Contact( "E105" )
      Contact( "TopEnd" )
      Contact( "M10.4" )
   END_RUNG wire#w3
   RUNG wire#w3
      R_Coil( "M5.6" )
   END_RUNG
   RUNG wire#w3
      R_Coil( "M5.4" )
   END_RUNG
   RUNG wire#w3
      R_Coil( "V89_5" )
   END_RUNG
   // the same network as SCL:
   IF ("M5.6" AND (("DB03_Machine".TopBefore AND "M0.1") OR ("DB03_Machine".TopWaterP AND "M3.3")) AND "Auto") OR ("M5.4" AND "E105" AND "TopEnd" AND "M10.4") THEN
       "M5.7" := TRUE;
   END_IF;
   #_w1 := ("M5.6" AND (("DB03_Machine".TopBefore AND "M0.1") OR ("DB03_Machine".TopWaterP AND "M3.3")) AND "Auto") OR ("M5.4" AND "E105" AND "TopEnd" AND "M10.4");
   IF #_w1 THEN
       "M5.6" := FALSE;
       "M5.4" := FALSE;
       "V89_5" := FALSE;
   END_IF;
END_REGION

REGION Network 56: Top cycle: M6.0 Start cycle
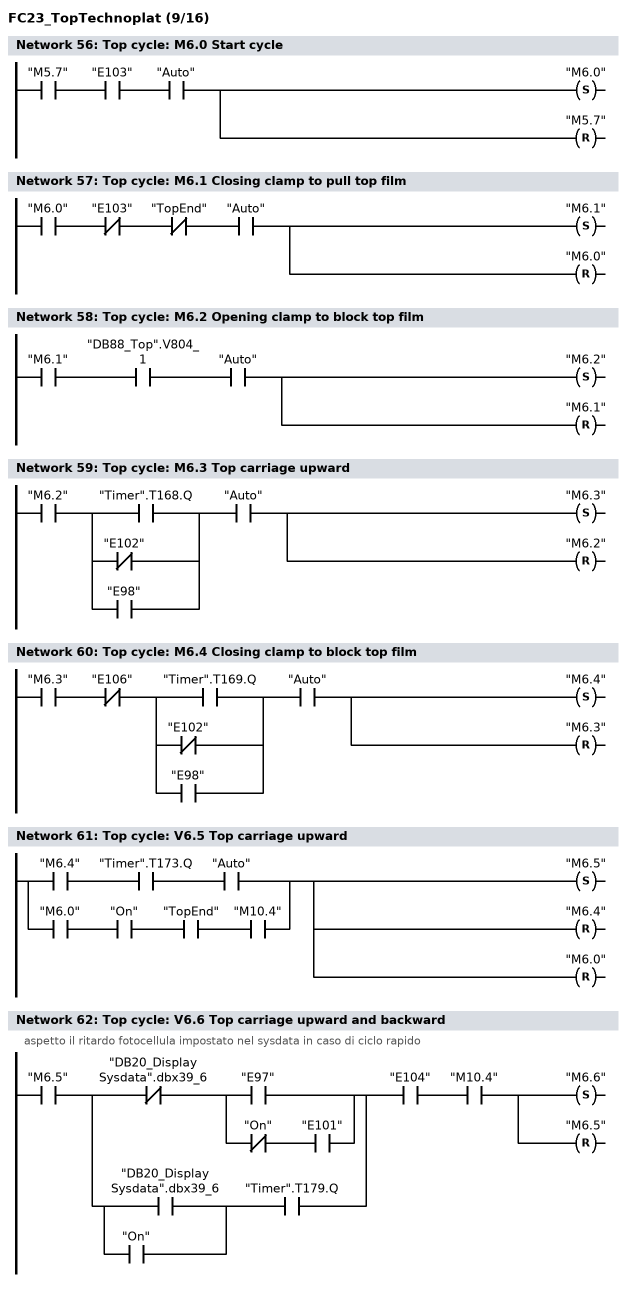
   RUNG wire#powerrail
      Contact( "M5.7" )
      Contact( "E103" )
      Contact( "Auto" )
      wire#w1
      S_Coil( "M6.0" )
   END_RUNG
   RUNG wire#w1
      R_Coil( "M5.7" )
   END_RUNG
   // the same network as SCL:
   IF "M5.7" AND "E103" AND "Auto" THEN
       "M6.0" := TRUE;
       "M5.7" := FALSE;
   END_IF;
END_REGION

REGION Network 57: Top cycle: M6.1 Closing clamp to pull top film
   RUNG wire#powerrail
      Contact( "M6.0" )
      I_Contact( "E103" )
      I_Contact( "TopEnd" )
      Contact( "Auto" )
      wire#w1
      S_Coil( "M6.1" )
   END_RUNG
   RUNG wire#w1
      R_Coil( "M6.0" )
   END_RUNG
   // the same network as SCL:
   IF "M6.0" AND NOT "E103" AND NOT "TopEnd" AND "Auto" THEN
       "M6.1" := TRUE;
       "M6.0" := FALSE;
   END_IF;
END_REGION

REGION Network 58: Top cycle: M6.2 Opening clamp to block top film
   RUNG wire#powerrail
      Contact( "M6.1" )
      Contact( "DB88_Top".V804_1 )
      Contact( "Auto" )
      wire#w1
      S_Coil( "M6.2" )
   END_RUNG
   RUNG wire#w1
      R_Coil( "M6.1" )
   END_RUNG
   // the same network as SCL:
   IF "M6.1" AND "DB88_Top".V804_1 AND "Auto" THEN
       "M6.2" := TRUE;
       "M6.1" := FALSE;
   END_IF;
END_REGION

REGION Network 59: Top cycle: M6.3 Top carriage upward
   RUNG wire#powerrail
      Contact( "M6.2" )
      wire#w1
      Contact( "Timer".T168.Q )
      wire#w2
      Contact( "Auto" )
      wire#w3
      S_Coil( "M6.3" )
   END_RUNG
   RUNG wire#w1
      I_Contact( "E102" )
   END_RUNG wire#w2
   RUNG wire#w1
      Contact( "E98" )
   END_RUNG wire#w2
   RUNG wire#w3
      R_Coil( "M6.2" )
   END_RUNG
   // the same network as SCL:
   IF "M6.2" AND ("Timer".T168.Q OR NOT "E102" OR "E98") AND "Auto" THEN
       "M6.3" := TRUE;
       "M6.2" := FALSE;
   END_IF;
END_REGION

REGION Network 60: Top cycle: M6.4 Closing clamp to block top film
   RUNG wire#powerrail
      Contact( "M6.3" )
      I_Contact( "E106" )
      wire#w1
      Contact( "Timer".T169.Q )
      wire#w2
      Contact( "Auto" )
      wire#w3
      S_Coil( "M6.4" )
   END_RUNG
   RUNG wire#w1
      I_Contact( "E102" )
   END_RUNG wire#w2
   RUNG wire#w1
      Contact( "E98" )
   END_RUNG wire#w2
   RUNG wire#w3
      R_Coil( "M6.3" )
   END_RUNG
   // the same network as SCL:
   IF "M6.3" AND NOT "E106" AND ("Timer".T169.Q OR NOT "E102" OR "E98") AND "Auto" THEN
       "M6.4" := TRUE;
       "M6.3" := FALSE;
   END_IF;
END_REGION

REGION Network 61: Top cycle: V6.5 Top carriage upward
   RUNG wire#powerrail
      Contact( "M6.4" )
      Contact( "Timer".T173.Q )
      Contact( "Auto" )
      wire#w1
      S_Coil( "M6.5" )
   END_RUNG
   RUNG wire#powerrail
      Contact( "M6.0" )
      Contact( "On" )
      Contact( "TopEnd" )
      Contact( "M10.4" )
   END_RUNG wire#w1
   RUNG wire#w1
      R_Coil( "M6.4" )
   END_RUNG
   RUNG wire#w1
      R_Coil( "M6.0" )
   END_RUNG
   // the same network as SCL:
   IF ("M6.4" AND "Timer".T173.Q AND "Auto") OR ("M6.0" AND "On" AND "TopEnd" AND "M10.4") THEN
       "M6.5" := TRUE;
   END_IF;
   #_w1 := ("M6.4" AND "Timer".T173.Q AND "Auto") OR ("M6.0" AND "On" AND "TopEnd" AND "M10.4");
   IF #_w1 THEN
       "M6.4" := FALSE;
       "M6.0" := FALSE;
   END_IF;
END_REGION

REGION Network 62: Top cycle: V6.6 Top carriage upward and backward
   // aspetto il ritardo fotocellula impostato nel sysdata in caso di ciclo rapido
   RUNG wire#powerrail
      Contact( "M6.5" )
      wire#w1
      I_Contact( "DB20_DisplaySysdata".dbx39_6 )
      wire#w2
      Contact( "E97" )
      wire#w3
      Contact( "E104" )
      Contact( "M10.4" )
      wire#w5
      S_Coil( "M6.6" )
   END_RUNG
   RUNG wire#w2
      I_Contact( "On" )
      Contact( "E101" )
   END_RUNG wire#w3
   RUNG wire#w1
      Contact( "DB20_DisplaySysdata".dbx39_6 )
      wire#w4
      Contact( "Timer".T179.Q )
   END_RUNG wire#w3
   RUNG wire#w1
      Contact( "On" )
   END_RUNG wire#w4
   RUNG wire#w5
      R_Coil( "M6.5" )
   END_RUNG
   // the same network as SCL:
   IF "M6.5" AND ((NOT "DB20_DisplaySysdata".dbx39_6 AND ("E97" OR (NOT "On" AND "E101"))) OR (("DB20_DisplaySysdata".dbx39_6 OR "On") AND "Timer".T179.Q)) AND "E104" AND "M10.4" THEN
       "M6.6" := TRUE;
       "M6.5" := FALSE;
   END_IF;
END_REGION

REGION Network 63: Top cycle: M6.7 Top cutter backward
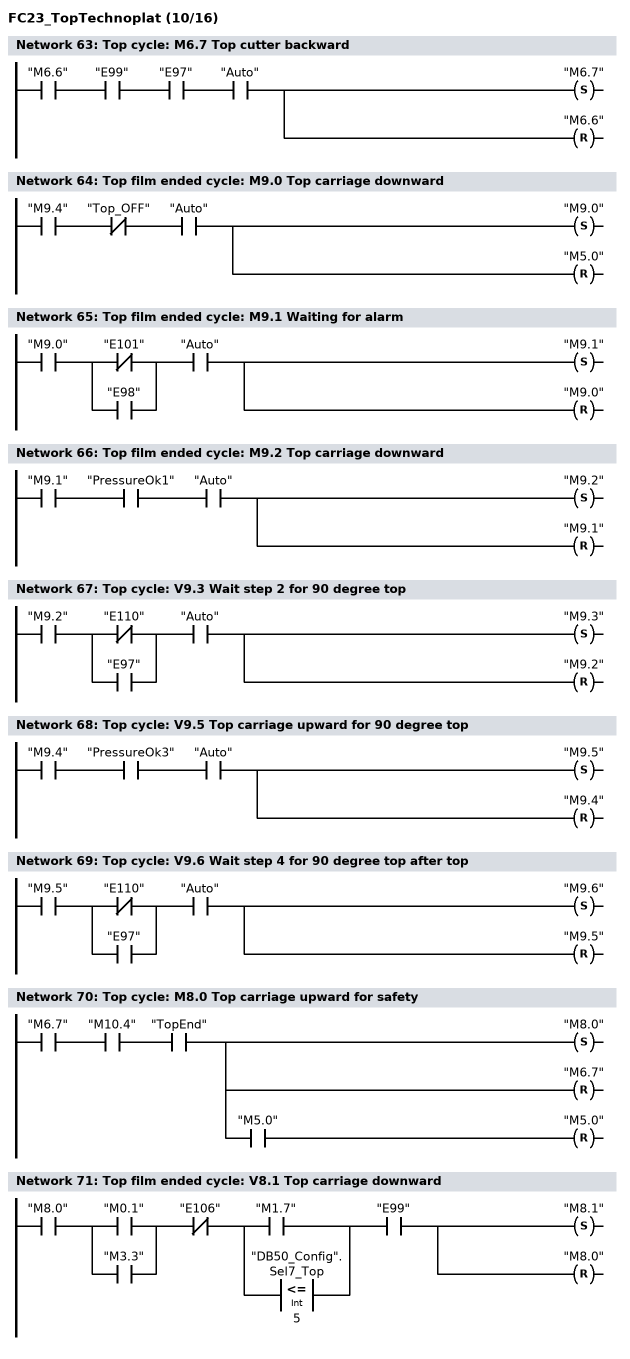
   RUNG wire#powerrail
      Contact( "M6.6" )
      Contact( "E99" )
      Contact( "E97" )
      Contact( "Auto" )
      wire#w1
      S_Coil( "M6.7" )
   END_RUNG
   RUNG wire#w1
      R_Coil( "M6.6" )
   END_RUNG
   // the same network as SCL:
   IF "M6.6" AND "E99" AND "E97" AND "Auto" THEN
       "M6.7" := TRUE;
       "M6.6" := FALSE;
   END_IF;
END_REGION

REGION Network 64: Top film ended cycle: M9.0 Top carriage downward
   RUNG wire#powerrail
      Contact( "M9.4" )
      I_Contact( "Top_OFF" )
      Contact( "Auto" )
      wire#w1
      S_Coil( "M9.0" )
   END_RUNG
   RUNG wire#w1
      R_Coil( "M5.0" )
   END_RUNG
   // the same network as SCL:
   IF "M9.4" AND NOT "Top_OFF" AND "Auto" THEN
       "M9.0" := TRUE;
       "M5.0" := FALSE;
   END_IF;
END_REGION

REGION Network 65: Top film ended cycle: M9.1 Waiting for alarm
   RUNG wire#powerrail
      Contact( "M9.0" )
      wire#w1
      I_Contact( "E101" )
      wire#w2
      Contact( "Auto" )
      wire#w3
      S_Coil( "M9.1" )
   END_RUNG
   RUNG wire#w1
      Contact( "E98" )
   END_RUNG wire#w2
   RUNG wire#w3
      R_Coil( "M9.0" )
   END_RUNG
   // the same network as SCL:
   IF "M9.0" AND (NOT "E101" OR "E98") AND "Auto" THEN
       "M9.1" := TRUE;
       "M9.0" := FALSE;
   END_IF;
END_REGION

REGION Network 66: Top film ended cycle: M9.2 Top carriage downward
   RUNG wire#powerrail
      Contact( "M9.1" )
      Contact( "PressureOk1" )
      Contact( "Auto" )
      wire#w1
      S_Coil( "M9.2" )
   END_RUNG
   RUNG wire#w1
      R_Coil( "M9.1" )
   END_RUNG
   // the same network as SCL:
   IF "M9.1" AND "PressureOk1" AND "Auto" THEN
       "M9.2" := TRUE;
       "M9.1" := FALSE;
   END_IF;
END_REGION

REGION Network 67: Top cycle: V9.3 Wait step 2 for 90 degree top
   RUNG wire#powerrail
      Contact( "M9.2" )
      wire#w1
      I_Contact( "E110" )
      wire#w2
      Contact( "Auto" )
      wire#w3
      S_Coil( "M9.3" )
   END_RUNG
   RUNG wire#w1
      Contact( "E97" )
   END_RUNG wire#w2
   RUNG wire#w3
      R_Coil( "M9.2" )
   END_RUNG
   // the same network as SCL:
   IF "M9.2" AND (NOT "E110" OR "E97") AND "Auto" THEN
       "M9.3" := TRUE;
       "M9.2" := FALSE;
   END_IF;
END_REGION

REGION Network 68: Top cycle: V9.5 Top carriage upward for 90 degree top
   RUNG wire#powerrail
      Contact( "M9.4" )
      Contact( "PressureOk3" )
      Contact( "Auto" )
      wire#w1
      S_Coil( "M9.5" )
   END_RUNG
   RUNG wire#w1
      R_Coil( "M9.4" )
   END_RUNG
   // the same network as SCL:
   IF "M9.4" AND "PressureOk3" AND "Auto" THEN
       "M9.5" := TRUE;
       "M9.4" := FALSE;
   END_IF;
END_REGION

REGION Network 69: Top cycle: V9.6 Wait step 4 for 90 degree top after top
   RUNG wire#powerrail
      Contact( "M9.5" )
      wire#w1
      I_Contact( "E110" )
      wire#w2
      Contact( "Auto" )
      wire#w3
      S_Coil( "M9.6" )
   END_RUNG
   RUNG wire#w1
      Contact( "E97" )
   END_RUNG wire#w2
   RUNG wire#w3
      R_Coil( "M9.5" )
   END_RUNG
   // the same network as SCL:
   IF "M9.5" AND (NOT "E110" OR "E97") AND "Auto" THEN
       "M9.6" := TRUE;
       "M9.5" := FALSE;
   END_IF;
END_REGION

REGION Network 70: Top cycle: M8.0 Top carriage upward for safety
   RUNG wire#powerrail
      Contact( "M6.7" )
      Contact( "M10.4" )
      Contact( "TopEnd" )
      wire#w1
      S_Coil( "M8.0" )
   END_RUNG
   RUNG wire#w1
      R_Coil( "M6.7" )
   END_RUNG
   RUNG wire#w1
      Contact( "M5.0" )
      R_Coil( "M5.0" )
   END_RUNG
   // the same network as SCL:
   #_w1 := "M6.7" AND "M10.4" AND "TopEnd";
   IF #_w1 THEN
       "M8.0" := TRUE;
       "M6.7" := FALSE;
   END_IF;
   IF #_w1 AND "M5.0" THEN "M5.0" := FALSE; END_IF;
END_REGION

REGION Network 71: Top film ended cycle: V8.1 Top carriage downward
   RUNG wire#powerrail
      Contact( "M8.0" )
      wire#w1
      Contact( "M0.1" )
      wire#w2
      I_Contact( "E106" )
      wire#w3
      Contact( "M1.7" )
      wire#w4
      Contact( "E99" )
      wire#w5
      S_Coil( "M8.1" )
   END_RUNG
   RUNG wire#w1
      Contact( "M3.3" )
   END_RUNG wire#w2
   RUNG wire#w3
      { S7_Templates := "SrcType := Int" } LE_Contact(in1 := "DB50_Config".Sel7_Top, in2 := 5)
   END_RUNG wire#w4
   RUNG wire#w5
      R_Coil( "M8.0" )
   END_RUNG
   // the same network as SCL:
   IF "M8.0" AND ("M0.1" OR "M3.3") AND NOT "E106" AND ("M1.7" OR ("DB50_Config".Sel7_Top <= 5)) AND "E99" THEN
       "M8.1" := TRUE;
       "M8.0" := FALSE;
   END_IF;
END_REGION

REGION Network 72: Top film ended cycle: V8.2 Top carriage forward
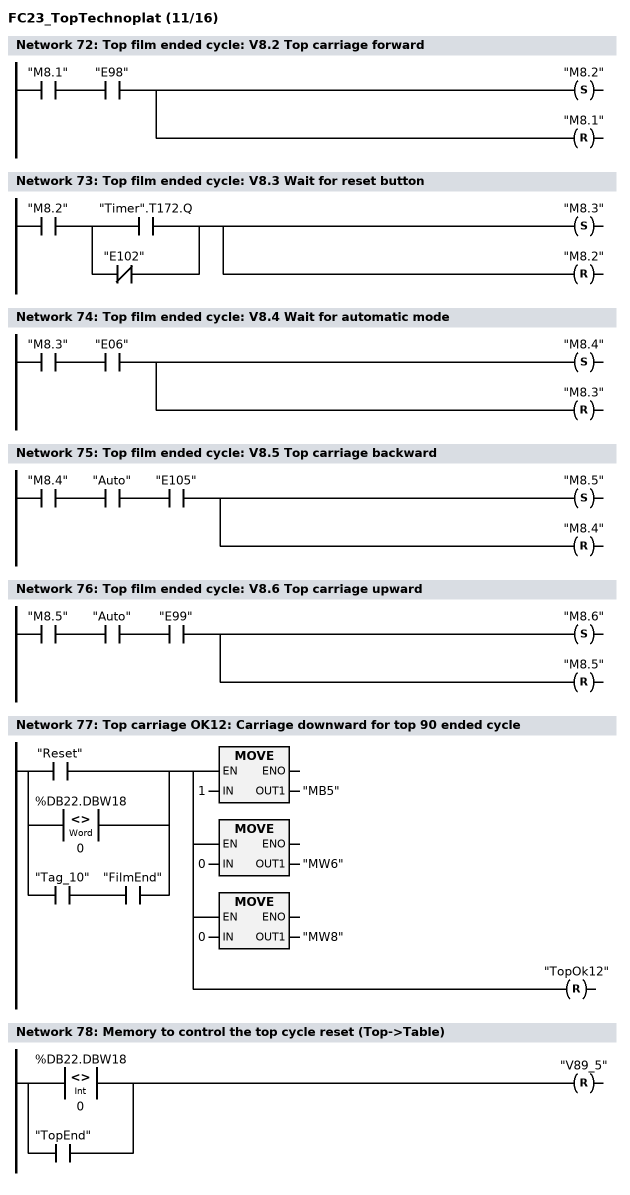
   RUNG wire#powerrail
      Contact( "M8.1" )
      Contact( "E98" )
      wire#w1
      S_Coil( "M8.2" )
   END_RUNG
   RUNG wire#w1
      R_Coil( "M8.1" )
   END_RUNG
   // the same network as SCL:
   IF "M8.1" AND "E98" THEN
       "M8.2" := TRUE;
       "M8.1" := FALSE;
   END_IF;
END_REGION

REGION Network 73: Top film ended cycle: V8.3 Wait for reset button
   RUNG wire#powerrail
      Contact( "M8.2" )
      wire#w1
      Contact( "Timer".T172.Q )
      wire#w2
      S_Coil( "M8.3" )
   END_RUNG
   RUNG wire#w1
      I_Contact( "E102" )
   END_RUNG wire#w2
   RUNG wire#w2
      R_Coil( "M8.2" )
   END_RUNG
   // the same network as SCL:
   IF "M8.2" AND ("Timer".T172.Q OR NOT "E102") THEN
       "M8.3" := TRUE;
       "M8.2" := FALSE;
   END_IF;
END_REGION

REGION Network 74: Top film ended cycle: V8.4 Wait for automatic mode
   RUNG wire#powerrail
      Contact( "M8.3" )
      Contact( "E06" )
      wire#w1
      S_Coil( "M8.4" )
   END_RUNG
   RUNG wire#w1
      R_Coil( "M8.3" )
   END_RUNG
   // the same network as SCL:
   IF "M8.3" AND "E06" THEN
       "M8.4" := TRUE;
       "M8.3" := FALSE;
   END_IF;
END_REGION

REGION Network 75: Top film ended cycle: V8.5 Top carriage backward
   RUNG wire#powerrail
      Contact( "M8.4" )
      Contact( "Auto" )
      Contact( "E105" )
      wire#w1
      S_Coil( "M8.5" )
   END_RUNG
   RUNG wire#w1
      R_Coil( "M8.4" )
   END_RUNG
   // the same network as SCL:
   IF "M8.4" AND "Auto" AND "E105" THEN
       "M8.5" := TRUE;
       "M8.4" := FALSE;
   END_IF;
END_REGION

REGION Network 76: Top film ended cycle: V8.6 Top carriage upward
   RUNG wire#powerrail
      Contact( "M8.5" )
      Contact( "Auto" )
      Contact( "E99" )
      wire#w1
      S_Coil( "M8.6" )
   END_RUNG
   RUNG wire#w1
      R_Coil( "M8.5" )
   END_RUNG
   // the same network as SCL:
   IF "M8.5" AND "Auto" AND "E99" THEN
       "M8.6" := TRUE;
       "M8.5" := FALSE;
   END_IF;
END_REGION

REGION Network 77: Top carriage OK12: Carriage downward for top 90 ended cycle
   RUNG wire#powerrail
      Contact( "Reset" )
      wire#w1
      { S7_GenerateENO := "TRUE" } Move(in := 1, out1 => "MB5")
   END_RUNG
   RUNG wire#powerrail
      { S7_Templates := "SrcType := Word" } NE_Contact(in1 := %DB22.DBW18, in2 := 0)
   END_RUNG wire#w1
   RUNG wire#powerrail
      Contact( "Tag_10" )
      Contact( "FilmEnd" )
   END_RUNG wire#w1
   RUNG wire#w1
      { S7_GenerateENO := "TRUE" } Move(in := 0, out1 => "MW6")
   END_RUNG
   RUNG wire#w1
      { S7_GenerateENO := "TRUE" } Move(in := 0, out1 => "MW8")
   END_RUNG
   RUNG wire#w1
      R_Coil( "TopOk12" )
   END_RUNG
   // the same network as SCL:
   IF "Reset" OR (%DB22.DBW18 <> 0) OR ("Tag_10" AND "FilmEnd") THEN
       "MB5" := 1;
       "MW6" := 0;
       "MW8" := 0;
       "TopOk12" := FALSE;
   END_IF;
END_REGION

REGION Network 78: Memory to control the top cycle reset (Top->Table)
   RUNG wire#powerrail
      { S7_Templates := "SrcType := Int" } NE_Contact(in1 := %DB22.DBW18, in2 := 0)
      wire#w1
      R_Coil( "V89_5" )
   END_RUNG
   RUNG wire#powerrail
      Contact( "TopEnd" )
   END_RUNG wire#w1
   // the same network as SCL:
   IF (%DB22.DBW18 <> 0) OR "TopEnd" THEN "V89_5" := FALSE; END_IF;
END_REGION

REGION Network 79: Top carriage forward (Top)
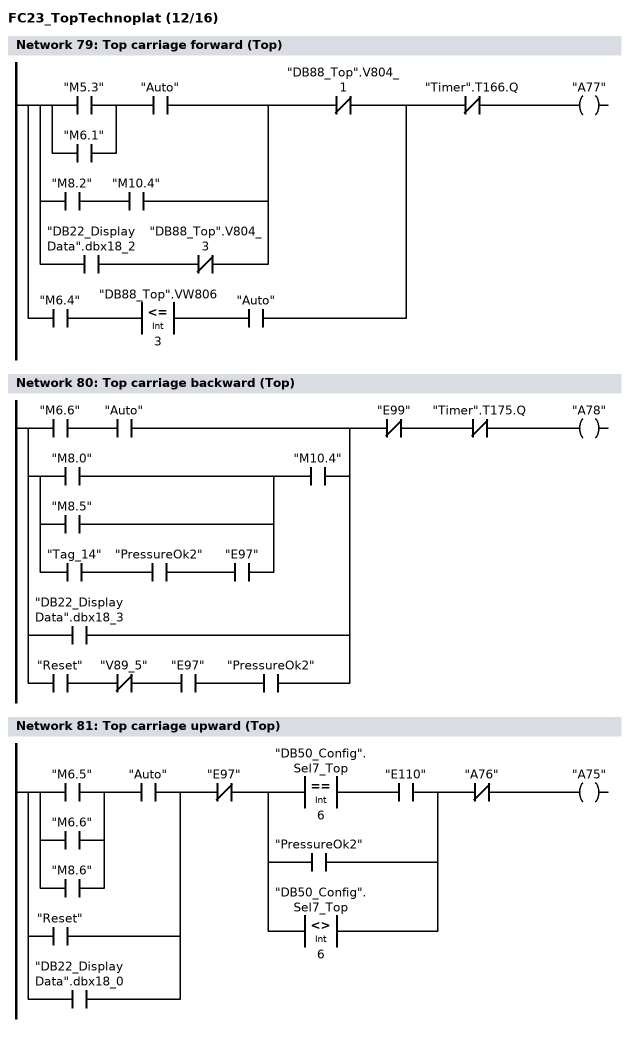
   RUNG wire#powerrail
      Contact( "M5.3" )
      wire#w1
      Contact( "Auto" )
      wire#w2
      I_Contact( "DB88_Top".V804_1 )
      wire#w3
      I_Contact( "Timer".T166.Q )
      Coil( "A77" )
   END_RUNG
   RUNG wire#powerrail
      Contact( "M6.1" )
   END_RUNG wire#w1
   RUNG wire#powerrail
      Contact( "M8.2" )
      Contact( "M10.4" )
   END_RUNG wire#w2
   RUNG wire#powerrail
      Contact( "DB22_DisplayData".dbx18_2 )
      I_Contact( "DB88_Top".V804_3 )
   END_RUNG wire#w2
   RUNG wire#powerrail
      Contact( "M6.4" )
      { S7_Templates := "SrcType := Int" } LE_Contact(in1 := "DB88_Top".VW806, in2 := 3)
      Contact( "Auto" )
   END_RUNG wire#w3
   // the same network as SCL:
   "A77" := ((((("M5.3" OR "M6.1") AND "Auto") OR ("M8.2" AND "M10.4") OR ("DB22_DisplayData".dbx18_2 AND NOT "DB88_Top".V804_3)) AND NOT "DB88_Top".V804_1) OR ("M6.4" AND ("DB88_Top".VW806 <= 3) AND "Auto")) AND NOT "Timer".T166.Q;
END_REGION

REGION Network 80: Top carriage backward (Top)
   RUNG wire#powerrail
      Contact( "M6.6" )
      Contact( "Auto" )
      wire#w1
      I_Contact( "E99" )
      I_Contact( "Timer".T175.Q )
      Coil( "A78" )
   END_RUNG
   RUNG wire#powerrail
      Contact( "M8.0" )
      wire#w2
      Contact( "M10.4" )
   END_RUNG wire#w1
   RUNG wire#powerrail
      Contact( "M8.5" )
   END_RUNG wire#w2
   RUNG wire#powerrail
      Contact( "Tag_14" )
      Contact( "PressureOk2" )
      Contact( "E97" )
   END_RUNG wire#w2
   RUNG wire#powerrail
      Contact( "DB22_DisplayData".dbx18_3 )
   END_RUNG wire#w1
   RUNG wire#powerrail
      Contact( "Reset" )
      I_Contact( "V89_5" )
      Contact( "E97" )
      Contact( "PressureOk2" )
   END_RUNG wire#w1
   // the same network as SCL:
   "A78" := (("M6.6" AND "Auto") OR (("M8.0" OR "M8.5" OR ("Tag_14" AND "PressureOk2" AND "E97")) AND "M10.4") OR "DB22_DisplayData".dbx18_3 OR ("Reset" AND NOT "V89_5" AND "E97" AND "PressureOk2")) AND NOT "E99" AND NOT "Timer".T175.Q;
END_REGION

REGION Network 81: Top carriage upward (Top)
   RUNG wire#powerrail
      Contact( "M6.5" )
      wire#w1
      Contact( "Auto" )
      wire#w2
      I_Contact( "E97" )
      wire#w3
      { S7_Templates := "SrcType := Int" } EQ_Contact(in1 := "DB50_Config".Sel7_Top, in2 := 6)
      Contact( "E110" )
      wire#w4
      I_Contact( "A76" )
      Coil( "A75" )
   END_RUNG
   RUNG wire#powerrail
      Contact( "M6.6" )
   END_RUNG wire#w1
   RUNG wire#powerrail
      Contact( "M8.6" )
   END_RUNG wire#w1
   RUNG wire#powerrail
      Contact( "Reset" )
   END_RUNG wire#w2
   RUNG wire#powerrail
      Contact( "DB22_DisplayData".dbx18_0 )
   END_RUNG wire#w2
   RUNG wire#w3
      Contact( "PressureOk2" )
   END_RUNG wire#w4
   RUNG wire#w3
      { S7_Templates := "SrcType := Int" } NE_Contact(in1 := "DB50_Config".Sel7_Top, in2 := 6)
   END_RUNG wire#w4
   // the same network as SCL:
   "A75" := ((("M6.5" OR "M6.6" OR "M8.6") AND "Auto") OR "Reset" OR "DB22_DisplayData".dbx18_0) AND NOT "E97" AND ((("DB50_Config".Sel7_Top = 6) AND "E110") OR "PressureOk2" OR ("DB50_Config".Sel7_Top <> 6)) AND NOT "A76";
END_REGION

REGION Network 82: Top carriage downward (Top)
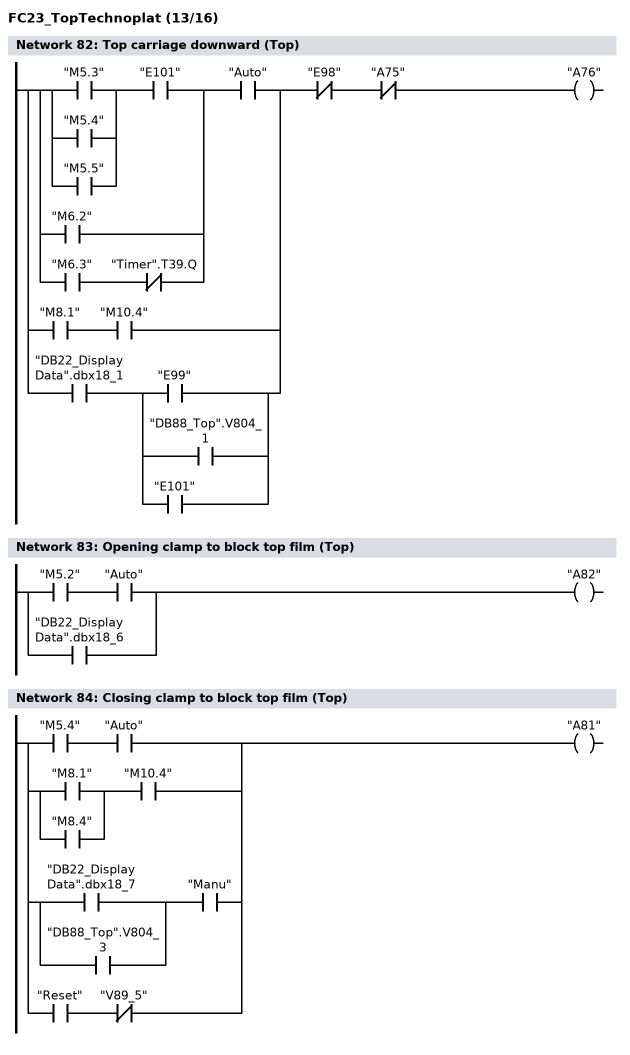
   RUNG wire#powerrail
      Contact( "M5.3" )
      wire#w1
      Contact( "E101" )
      wire#w2
      Contact( "Auto" )
      wire#w3
      I_Contact( "E98" )
      I_Contact( "A75" )
      Coil( "A76" )
   END_RUNG
   RUNG wire#powerrail
      Contact( "M5.4" )
   END_RUNG wire#w1
   RUNG wire#powerrail
      Contact( "M5.5" )
   END_RUNG wire#w1
   RUNG wire#powerrail
      Contact( "M6.2" )
   END_RUNG wire#w2
   RUNG wire#powerrail
      Contact( "M6.3" )
      I_Contact( "Timer".T39.Q )
   END_RUNG wire#w2
   RUNG wire#powerrail
      Contact( "M8.1" )
      Contact( "M10.4" )
   END_RUNG wire#w3
   RUNG wire#powerrail
      Contact( "DB22_DisplayData".dbx18_1 )
      wire#w4
      Contact( "E99" )
   END_RUNG wire#w3
   RUNG wire#w4
      Contact( "DB88_Top".V804_1 )
   END_RUNG wire#w3
   RUNG wire#w4
      Contact( "E101" )
   END_RUNG wire#w3
   // the same network as SCL:
   "A76" := ((((("M5.3" OR "M5.4" OR "M5.5") AND "E101") OR "M6.2" OR ("M6.3" AND NOT "Timer".T39.Q)) AND "Auto") OR ("M8.1" AND "M10.4") OR ("DB22_DisplayData".dbx18_1 AND ("E99" OR "DB88_Top".V804_1 OR "E101"))) AND NOT "E98" AND NOT "A75";
END_REGION

REGION Network 83: Opening clamp to block top film (Top)
   RUNG wire#powerrail
      Contact( "M5.2" )
      Contact( "Auto" )
      wire#w1
      Coil( "A82" )
   END_RUNG
   RUNG wire#powerrail
      Contact( "DB22_DisplayData".dbx18_6 )
   END_RUNG wire#w1
   // the same network as SCL:
   "A82" := ("M5.2" AND "Auto") OR "DB22_DisplayData".dbx18_6;
END_REGION

REGION Network 84: Closing clamp to block top film (Top)
   RUNG wire#powerrail
      Contact( "M5.4" )
      Contact( "Auto" )
      wire#w1
      Coil( "A81" )
   END_RUNG
   RUNG wire#powerrail
      Contact( "M8.1" )
      wire#w2
      Contact( "M10.4" )
   END_RUNG wire#w1
   RUNG wire#powerrail
      Contact( "M8.4" )
   END_RUNG wire#w2
   RUNG wire#powerrail
      Contact( "DB22_DisplayData".dbx18_7 )
      wire#w3
      Contact( "Manu" )
   END_RUNG wire#w1
   RUNG wire#powerrail
      Contact( "DB88_Top".V804_3 )
   END_RUNG wire#w3
   RUNG wire#powerrail
      Contact( "Reset" )
      I_Contact( "V89_5" )
   END_RUNG wire#w1
   // the same network as SCL:
   "A81" := ("M5.4" AND "Auto") OR (("M8.1" OR "M8.4") AND "M10.4") OR (("DB22_DisplayData".dbx18_7 OR "DB88_Top".V804_3) AND "Manu") OR ("Reset" AND NOT "V89_5");
END_REGION

REGION Network 85: Opening clamp to lift(pull) top film (Top)
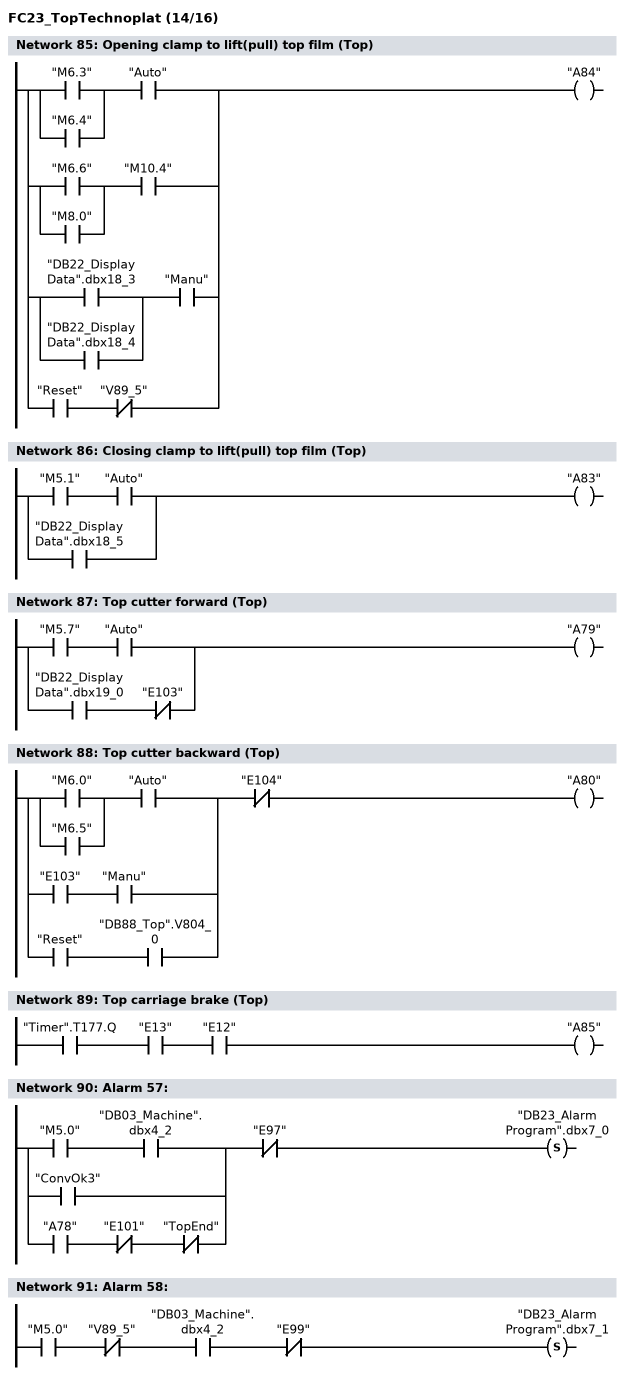
   RUNG wire#powerrail
      Contact( "M6.3" )
      wire#w1
      Contact( "Auto" )
      wire#w2
      Coil( "A84" )
   END_RUNG
   RUNG wire#powerrail
      Contact( "M6.4" )
   END_RUNG wire#w1
   RUNG wire#powerrail
      Contact( "M6.6" )
      wire#w3
      Contact( "M10.4" )
   END_RUNG wire#w2
   RUNG wire#powerrail
      Contact( "M8.0" )
   END_RUNG wire#w3
   RUNG wire#powerrail
      Contact( "DB22_DisplayData".dbx18_3 )
      wire#w4
      Contact( "Manu" )
   END_RUNG wire#w2
   RUNG wire#powerrail
      Contact( "DB22_DisplayData".dbx18_4 )
   END_RUNG wire#w4
   RUNG wire#powerrail
      Contact( "Reset" )
      I_Contact( "V89_5" )
   END_RUNG wire#w2
   // the same network as SCL:
   "A84" := (("M6.3" OR "M6.4") AND "Auto") OR (("M6.6" OR "M8.0") AND "M10.4") OR (("DB22_DisplayData".dbx18_3 OR "DB22_DisplayData".dbx18_4) AND "Manu") OR ("Reset" AND NOT "V89_5");
END_REGION

REGION Network 86: Closing clamp to lift(pull) top film (Top)
   RUNG wire#powerrail
      Contact( "M5.1" )
      Contact( "Auto" )
      wire#w1
      Coil( "A83" )
   END_RUNG
   RUNG wire#powerrail
      Contact( "DB22_DisplayData".dbx18_5 )
   END_RUNG wire#w1
   // the same network as SCL:
   "A83" := ("M5.1" AND "Auto") OR "DB22_DisplayData".dbx18_5;
END_REGION

REGION Network 87: Top cutter forward (Top)
   RUNG wire#powerrail
      Contact( "M5.7" )
      Contact( "Auto" )
      wire#w1
      Coil( "A79" )
   END_RUNG
   RUNG wire#powerrail
      Contact( "DB22_DisplayData".dbx19_0 )
      I_Contact( "E103" )
   END_RUNG wire#w1
   // the same network as SCL:
   "A79" := ("M5.7" AND "Auto") OR ("DB22_DisplayData".dbx19_0 AND NOT "E103");
END_REGION

REGION Network 88: Top cutter backward (Top)
   RUNG wire#powerrail
      Contact( "M6.0" )
      wire#w1
      Contact( "Auto" )
      wire#w2
      I_Contact( "E104" )
      Coil( "A80" )
   END_RUNG
   RUNG wire#powerrail
      Contact( "M6.5" )
   END_RUNG wire#w1
   RUNG wire#powerrail
      Contact( "E103" )
      Contact( "Manu" )
   END_RUNG wire#w2
   RUNG wire#powerrail
      Contact( "Reset" )
      Contact( "DB88_Top".V804_0 )
   END_RUNG wire#w2
   // the same network as SCL:
   "A80" := ((("M6.0" OR "M6.5") AND "Auto") OR ("E103" AND "Manu") OR ("Reset" AND "DB88_Top".V804_0)) AND NOT "E104";
END_REGION

REGION Network 89: Top carriage brake (Top)
   RUNG wire#powerrail
      Contact( "Timer".T177.Q )
      Contact( "E13" )
      Contact( "E12" )
      Coil( "A85" )
   END_RUNG
   // the same network as SCL:
   "A85" := "Timer".T177.Q AND "E13" AND "E12";
END_REGION

REGION Network 90: Alarm 57:
   RUNG wire#powerrail
      Contact( "M5.0" )
      Contact( "DB03_Machine".dbx4_2 )
      wire#w1
      I_Contact( "E97" )
      S_Coil( "DB23_AlarmProgram".dbx7_0 )
   END_RUNG
   RUNG wire#powerrail
      Contact( "ConvOk3" )
   END_RUNG wire#w1
   RUNG wire#powerrail
      Contact( "A78" )
      I_Contact( "E101" )
      I_Contact( "TopEnd" )
   END_RUNG wire#w1
   // the same network as SCL:
   IF (("M5.0" AND "DB03_Machine".dbx4_2) OR "ConvOk3" OR ("A78" AND NOT "E101" AND NOT "TopEnd")) AND NOT "E97" THEN
       "DB23_AlarmProgram".dbx7_0 := TRUE;
   END_IF;
END_REGION

REGION Network 91: Alarm 58:
   RUNG wire#powerrail
      Contact( "M5.0" )
      I_Contact( "V89_5" )
      Contact( "DB03_Machine".dbx4_2 )
      I_Contact( "E99" )
      S_Coil( "DB23_AlarmProgram".dbx7_1 )
   END_RUNG
   // the same network as SCL:
   IF "M5.0" AND NOT "V89_5" AND "DB03_Machine".dbx4_2 AND NOT "E99" THEN
       "DB23_AlarmProgram".dbx7_1 := TRUE;
   END_IF;
END_REGION

REGION Network 92: Alarm 59:
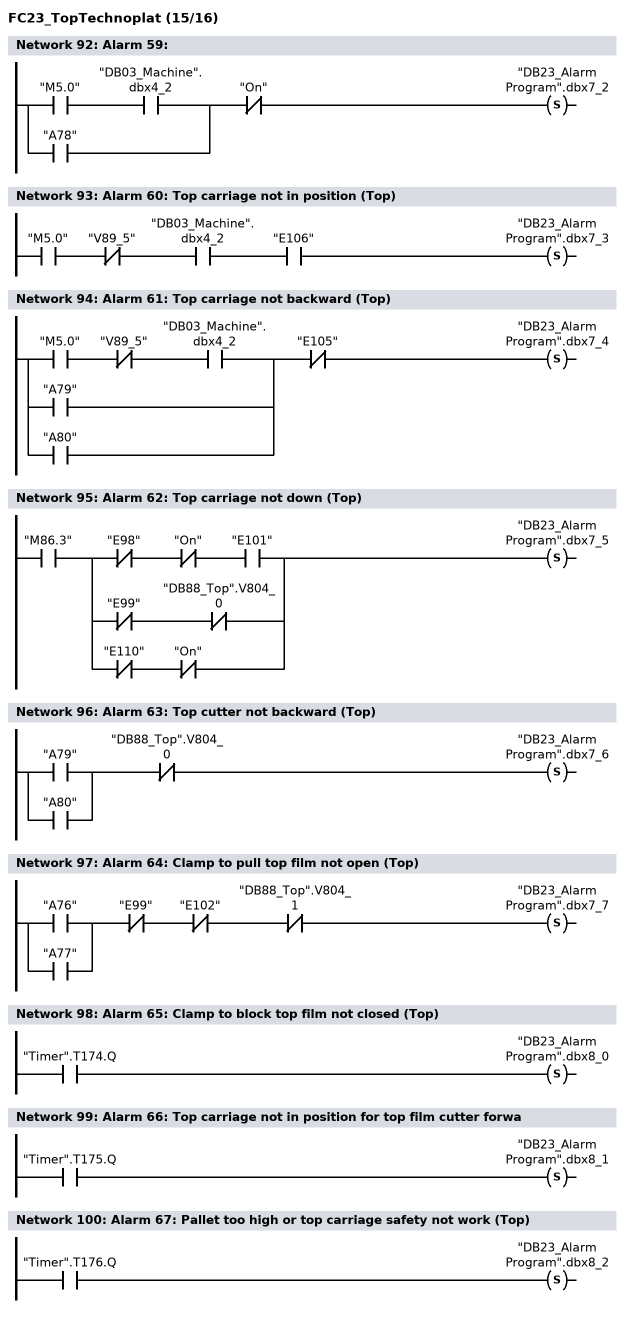
   RUNG wire#powerrail
      Contact( "M5.0" )
      Contact( "DB03_Machine".dbx4_2 )
      wire#w1
      I_Contact( "On" )
      S_Coil( "DB23_AlarmProgram".dbx7_2 )
   END_RUNG
   RUNG wire#powerrail
      Contact( "A78" )
   END_RUNG wire#w1
   // the same network as SCL:
   IF (("M5.0" AND "DB03_Machine".dbx4_2) OR "A78") AND NOT "On" THEN
       "DB23_AlarmProgram".dbx7_2 := TRUE;
   END_IF;
END_REGION

REGION Network 93: Alarm 60: Top carriage not in position (Top)
   RUNG wire#powerrail
      Contact( "M5.0" )
      I_Contact( "V89_5" )
      Contact( "DB03_Machine".dbx4_2 )
      Contact( "E106" )
      S_Coil( "DB23_AlarmProgram".dbx7_3 )
   END_RUNG
   // the same network as SCL:
   IF "M5.0" AND NOT "V89_5" AND "DB03_Machine".dbx4_2 AND "E106" THEN
       "DB23_AlarmProgram".dbx7_3 := TRUE;
   END_IF;
END_REGION

REGION Network 94: Alarm 61: Top carriage not backward (Top)
   RUNG wire#powerrail
      Contact( "M5.0" )
      I_Contact( "V89_5" )
      Contact( "DB03_Machine".dbx4_2 )
      wire#w1
      I_Contact( "E105" )
      S_Coil( "DB23_AlarmProgram".dbx7_4 )
   END_RUNG
   RUNG wire#powerrail
      Contact( "A79" )
   END_RUNG wire#w1
   RUNG wire#powerrail
      Contact( "A80" )
   END_RUNG wire#w1
   // the same network as SCL:
   IF (("M5.0" AND NOT "V89_5" AND "DB03_Machine".dbx4_2) OR "A79" OR "A80") AND NOT "E105" THEN
       "DB23_AlarmProgram".dbx7_4 := TRUE;
   END_IF;
END_REGION

REGION Network 95: Alarm 62: Top carriage not down (Top)
   RUNG wire#powerrail
      Contact( "M86.3" )
      wire#w1
      I_Contact( "E98" )
      I_Contact( "On" )
      Contact( "E101" )
      wire#w2
      S_Coil( "DB23_AlarmProgram".dbx7_5 )
   END_RUNG
   RUNG wire#w1
      I_Contact( "E99" )
      I_Contact( "DB88_Top".V804_0 )
   END_RUNG wire#w2
   RUNG wire#w1
      I_Contact( "E110" )
      I_Contact( "On" )
   END_RUNG wire#w2
   // the same network as SCL:
   IF "M86.3" AND ((NOT "E98" AND NOT "On" AND "E101") OR (NOT "E99" AND NOT "DB88_Top".V804_0) OR (NOT "E110" AND NOT "On")) THEN
       "DB23_AlarmProgram".dbx7_5 := TRUE;
   END_IF;
END_REGION

REGION Network 96: Alarm 63: Top cutter not backward (Top)
   RUNG wire#powerrail
      Contact( "A79" )
      wire#w1
      I_Contact( "DB88_Top".V804_0 )
      S_Coil( "DB23_AlarmProgram".dbx7_6 )
   END_RUNG
   RUNG wire#powerrail
      Contact( "A80" )
   END_RUNG wire#w1
   // the same network as SCL:
   IF ("A79" OR "A80") AND NOT "DB88_Top".V804_0 THEN "DB23_AlarmProgram".dbx7_6 := TRUE; END_IF;
END_REGION

REGION Network 97: Alarm 64: Clamp to pull top film not open (Top)
   RUNG wire#powerrail
      Contact( "A76" )
      wire#w1
      I_Contact( "E99" )
      I_Contact( "E102" )
      I_Contact( "DB88_Top".V804_1 )
      S_Coil( "DB23_AlarmProgram".dbx7_7 )
   END_RUNG
   RUNG wire#powerrail
      Contact( "A77" )
   END_RUNG wire#w1
   // the same network as SCL:
   IF ("A76" OR "A77") AND NOT "E99" AND NOT "E102" AND NOT "DB88_Top".V804_1 THEN
       "DB23_AlarmProgram".dbx7_7 := TRUE;
   END_IF;
END_REGION

REGION Network 98: Alarm 65: Clamp to block top film not closed (Top)
   RUNG wire#powerrail
      Contact( "Timer".T174.Q )
      S_Coil( "DB23_AlarmProgram".dbx8_0 )
   END_RUNG
   // the same network as SCL:
   IF "Timer".T174.Q THEN "DB23_AlarmProgram".dbx8_0 := TRUE; END_IF;
END_REGION

REGION Network 99: Alarm 66: Top carriage not in position for top film cutter forwa
   RUNG wire#powerrail
      Contact( "Timer".T175.Q )
      S_Coil( "DB23_AlarmProgram".dbx8_1 )
   END_RUNG
   // the same network as SCL:
   IF "Timer".T175.Q THEN "DB23_AlarmProgram".dbx8_1 := TRUE; END_IF;
END_REGION

REGION Network 100: Alarm 67: Pallet too high or top carriage safety not work (Top)
   RUNG wire#powerrail
      Contact( "Timer".T176.Q )
      S_Coil( "DB23_AlarmProgram".dbx8_2 )
   END_RUNG
   // the same network as SCL:
   IF "Timer".T176.Q THEN "DB23_AlarmProgram".dbx8_2 := TRUE; END_IF;
END_REGION

REGION Network 101: Alarm 68: Pallet too low or top carriage pallet height not work
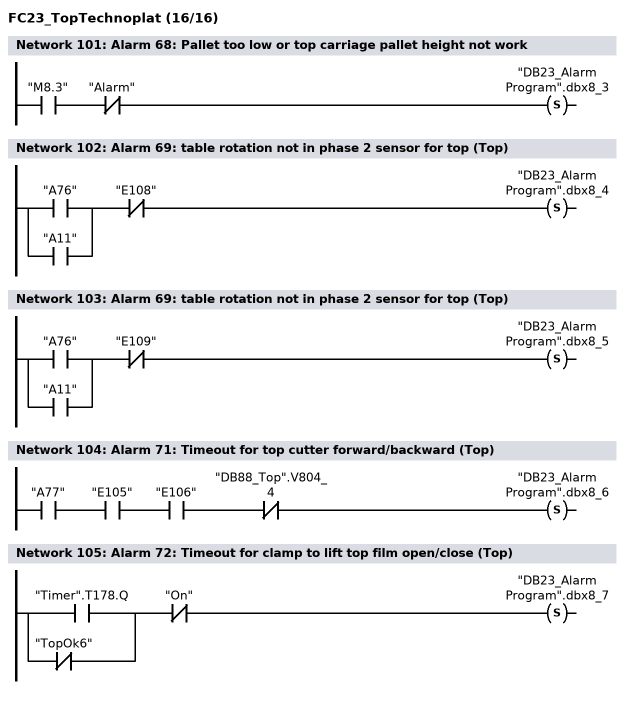
   RUNG wire#powerrail
      Contact( "M8.3" )
      I_Contact( "Alarm" )
      S_Coil( "DB23_AlarmProgram".dbx8_3 )
   END_RUNG
   // the same network as SCL:
   IF "M8.3" AND NOT "Alarm" THEN "DB23_AlarmProgram".dbx8_3 := TRUE; END_IF;
END_REGION

REGION Network 102: Alarm 69: table rotation not in phase 2 sensor for top (Top)
   RUNG wire#powerrail
      Contact( "A76" )
      wire#w1
      I_Contact( "E108" )
      S_Coil( "DB23_AlarmProgram".dbx8_4 )
   END_RUNG
   RUNG wire#powerrail
      Contact( "A11" )
   END_RUNG wire#w1
   // the same network as SCL:
   IF ("A76" OR "A11") AND NOT "E108" THEN "DB23_AlarmProgram".dbx8_4 := TRUE; END_IF;
END_REGION

REGION Network 103: Alarm 69: table rotation not in phase 2 sensor for top (Top)
   RUNG wire#powerrail
      Contact( "A76" )
      wire#w1
      I_Contact( "E109" )
      S_Coil( "DB23_AlarmProgram".dbx8_5 )
   END_RUNG
   RUNG wire#powerrail
      Contact( "A11" )
   END_RUNG wire#w1
   // the same network as SCL:
   IF ("A76" OR "A11") AND NOT "E109" THEN "DB23_AlarmProgram".dbx8_5 := TRUE; END_IF;
END_REGION

REGION Network 104: Alarm 71: Timeout for top cutter forward/backward (Top)
   RUNG wire#powerrail
      Contact( "A77" )
      Contact( "E105" )
      Contact( "E106" )
      I_Contact( "DB88_Top".V804_4 )
      S_Coil( "DB23_AlarmProgram".dbx8_6 )
   END_RUNG
   // the same network as SCL:
   IF "A77" AND "E105" AND "E106" AND NOT "DB88_Top".V804_4 THEN "DB23_AlarmProgram".dbx8_6 := TRUE; END_IF;
END_REGION

REGION Network 105: Alarm 72: Timeout for clamp to lift top film open/close (Top)
   RUNG wire#powerrail
      Contact( "Timer".T178.Q )
      wire#w1
      I_Contact( "On" )
      S_Coil( "DB23_AlarmProgram".dbx8_7 )
   END_RUNG
   RUNG wire#powerrail
      I_Contact( "TopOk6" )
   END_RUNG wire#w1
   // the same network as SCL:
   IF ("Timer".T178.Q OR NOT "TopOk6") AND NOT "On" THEN "DB23_AlarmProgram".dbx8_7 := TRUE; END_IF;
END_REGION
END_FUNCTION
